LIN {X 0,Y 525.492,Z 369.575,A -85,B 0,C 180,E1 -4793.237,E2 -4793.237} C_VEL
LIN {X 0,Y 523.983,Z 361.217,A -85,B 0,C 180,E1 -4794.674,E2 -4794.674} C_VEL
LIN {X 0,Y 523.979,Z 361.219,A -85,B 0,C 180,E1 -4797.718,E2 -4797.718} C_VEL
LIN {X 0,Y 523.947,Z 361.217,A -85,B 0,C 180,E1 -4800.855,E2 -4800.855} C_VEL
LIN {X 0,Y 523.96,Z 361.222,A -85,B 0,C 180,E1 -4803.734,E2 -4803.734} C_VEL
LIN {X 0,Y 523.921,Z 361.218,A -85,B 0,C 180,E1 -4806.404,E2 -4806.404} C_VEL
LIN {X 0,Y 523.921,Z 361.22,A -85,B 0,C 180,E1 -4809.084,E2 -4809.084} C_VEL
LIN {X 0,Y 523.954,Z 361.216,A -85,B 0,C 180,E1 -4812.118,E2 -4812.118} C_VEL
LIN {X 0,Y 523.952,Z 361.219,A -85,B 0,C 180,E1 -4815.308,E2 -4815.308} C_VEL
LIN {X 0,Y 523.968,Z 361.212,A -85,B 0,C 180,E1 -4818.687,E2 -4818.687} C_VEL
LIN {X 0,Y 523.92,Z 361.221,A -85,B 0,C 180,E1 -4821.079,E2 -4821.079} C_VEL
LIN {X 0,Y 523.922,Z 361.221,A -85,B 0,C 180,E1 -4823.827,E2 -4823.827} C_VEL
LIN {X 0,Y 523.937,Z 361.216,A -85,B 0,C 180,E1 -4826.635,E2 -4826.635} C_VEL
LIN {X 0,Y 523.957,Z 361.223,A -85,B 0,C 180,E1 -4829.356,E2 -4829.356} C_VEL
LIN {X 0,Y 523.973,Z 361.211,A -85,B 0,C 180,E1 -4832.28,E2 -4832.28} C_VEL
LIN {X 0,Y 523.948,Z 361.215,A -85,B 0,C 180,E1 -4834.581,E2 -4834.581} C_VEL
LIN {X 0,Y 523.937,Z 361.223,A -85,B 0,C 180,E1 -4837.108,E2 -4837.108} C_VEL
LIN {X 0,Y 523.971,Z 361.213,A -85,B 0,C 180,E1 -4839.865,E2 -4839.865} C_VEL
LIN {X 0,Y 523.963,Z 361.217,A -85,B 0,C 180,E1 -4842.837,E2 -4842.837} C_VEL
LIN {X 0,Y 523.967,Z 361.22,A -85,B 0,C 180,E1 -4845.235,E2 -4845.235} C_VEL
LIN {X 0,Y 524.004,Z 361.208,A -85,B 0,C 180,E1 -4848.394,E2 -4848.394} C_VEL
LIN {X 0,Y 524,Z 361.211,A -85,B 0,C 180,E1 -4851.516,E2 -4851.516} C_VEL
LIN {X 0,Y 524.078,Z 361.202,A -85,B 0,C 180,E1 -4854.614,E2 -4854.614} C_VEL
LIN {X 0,Y 524.104,Z 361.196,A -85,B 0,C 180,E1 -4857.694,E2 -4857.694} C_VEL
LIN {X 0,Y 524.119,Z 361.2,A -85,B 0,C 180,E1 -4860.768,E2 -4860.768} C_VEL
LIN {X 0,Y 524.07,Z 361.206,A -85,B 0,C 180,E1 -4863.075,E2 -4863.075} C_VEL
LIN {X 0,Y 524.038,Z 361.204,A -85,B 0,C 180,E1 -4866.159,E2 -4866.159} C_VEL
LIN {X 0,Y 523.996,Z 361.211,A -85,B 0,C 180,E1 -4869.262,E2 -4869.262} C_VEL
LIN {X 0,Y 524.015,Z 361.206,A -85,B 0,C 180,E1 -4871.752,E2 -4871.752} C_VEL
LIN {X 0,Y 523.984,Z 361.214,A -85,B 0,C 180,E1 -4875.053,E2 -4875.053} C_VEL
LIN {X 0,Y 523.956,Z 361.214,A -85,B 0,C 180,E1 -4877.969,E2 -4877.969} C_VEL
LIN {X 0,Y 523.965,Z 361.218,A -85,B 0,C 180,E1 -4880.41,E2 -4880.41} C_VEL
LIN {X 0,Y 523.937,Z 361.221,A -85,B 0,C 180,E1 -4882.893,E2 -4882.893} C_VEL
LIN {X 0,Y 523.978,Z 361.212,A -85,B 0,C 180,E1 -4886.021,E2 -4886.021} C_VEL
LIN {X 0,Y 523.934,Z 361.221,A -85,B 0,C 180,E1 -4888.875,E2 -4888.875} C_VEL
LIN {X 0,Y 523.925,Z 361.217,A -85,B 0,C 180,E1 -4891.544,E2 -4891.544} C_VEL
LIN {X 0,Y 523.934,Z 361.223,A -85,B 0,C 180,E1 -4894.29,E2 -4894.29} C_VEL
LIN {X 0,Y 523.906,Z 361.22,A -85,B 0,C 180,E1 -4897.133,E2 -4897.133} C_VEL
LIN {X 0,Y 523.963,Z 361.218,A -85,B 0,C 180,E1 -4900.135,E2 -4900.135} C_VEL
LIN {X 0,Y 523.922,Z 361.218,A -85,B 0,C 180,E1 -4903.167,E2 -4903.167} C_VEL
LIN {X 0,Y 523.935,Z 361.218,A -85,B 0,C 180,E1 -4905.773,E2 -4905.773} C_VEL
LIN {X 0,Y 523.913,Z 361.22,A -85,B 0,C 180,E1 -4906.931,E2 -4906.931} C_VEL
LIN {X 0,Y 523.248,Z 361.303,A -85,B 0,C 180,E1 -4907.572,E2 -4907.572} C_VEL
LIN {X 0,Y 520.406,Z 361.666,A -85,B 0,C 180,E1 -4908.614,E2 -4908.614} C_VEL
LIN {X 0,Y 518,Z 361.971,A -85,B 0,C 180,E1 -4909.453,E2 -4909.453} C_VEL
LIN {X 0,Y 516.965,Z 362.096,A -85,B 0,C 180,E1 -4910.101,E2 -4910.101} C_VEL
LIN {X 0,Y 516.879,Z 362.103,A -85,B 0,C 180,E1 -4910.32,E2 -4910.32} C_VEL
LIN {X 0,Y 516.884,Z 362.095,A -85,B 0,C 180,E1 -4913.343,E2 -4913.343} C_VEL
LIN {X 0,Y 516.911,Z 362.1,A -85,B 0,C 180,E1 -4916.122,E2 -4916.122} C_VEL
LIN {X 0,Y 516.892,Z 362.094,A -85,B 0,C 180,E1 -4918.936,E2 -4918.936} C_VEL
LIN {X 0,Y 516.92,Z 362.092,A -85,B 0,C 180,E1 -4921.586,E2 -4921.586} C_VEL
LIN {X 0,Y 516.93,Z 362.097,A -85,B 0,C 180,E1 -4924.212,E2 -4924.212} C_VEL
LIN {X 0,Y 516.861,Z 362.101,A -85,B 0,C 180,E1 -4926.777,E2 -4926.777} C_VEL
LIN {X 0,Y 516.963,Z 362.173,A -85,B 0,C 180,E1 -4929.932,E2 -4929.932} C_VEL
LIN {X 0,Y 517.701,Z 368.131,A -85,B 0,C 180,E1 -4931.191,E2 -4931.191} C_VEL
LIN {X 0,Y 517.28,Z 383.258,A -85,B 0,C 180,E1 -4934.233,E2 -4934.233} C_VEL
LIN {X 0,Y 517.249,Z 385.513,A -85,B 0,C 180,E1 -4934.682,E2 -4934.682} C_VEL
LIN {X 0,Y 519.15,Z 395.792,A -85,B 0,C 180,E1 -4934.899,E2 -4934.899} C_VEL
LIN {X 0,Y 518.657,Z 492.288,A -85,B 0,C 180,E1 -4936.258,E2 -4936.258} C_VEL
LIN {X 0,Y 518.471,Z 505.449,A -85,B 0,C 180,E1 -4936.603,E2 -4936.603} C_VEL
LIN {X 0,Y 518.233,Z 517.533,A -85,B 0,C 180,E1 -4937.07,E2 -4937.07} C_VEL
LIN {X 0,Y 518.027,Z 528.523,A -85,B 0,C 180,E1 -4937.639,E2 -4937.639} C_VEL
LIN {X 0,Y 517.731,Z 539.307,A -85,B 0,C 180,E1 -4938.351,E2 -4938.351} C_VEL
LIN {X 0,Y 517.367,Z 549.993,A -85,B 0,C 180,E1 -4939.235,E2 -4939.235} C_VEL
LIN {X 0,Y 517.115,Z 559.603,A -85,B 0,C 180,E1 -4940.219,E2 -4940.219} C_VEL
LIN {X 0,Y 516.861,Z 567.474,A -85,B 0,C 180,E1 -4941.201,E2 -4941.201} C_VEL
LIN {X 0,Y 516.638,Z 575.169,A -85,B 0,C 180,E1 -4942.378,E2 -4942.378} C_VEL
LIN {X 0,Y 516.496,Z 582.223,A -85,B 0,C 180,E1 -4943.751,E2 -4943.751} C_VEL
LIN {X 0,Y 516.314,Z 586.928,A -85,B 0,C 180,E1 -4944.924,E2 -4944.924} C_VEL
LIN {X 0,Y 516.373,Z 590.524,A -85,B 0,C 180,E1 -4946.098,E2 -4946.098} C_VEL
LIN {X 0,Y 516.282,Z 592.387,A -85,B 0,C 180,E1 -4946.879,E2 -4946.879} C_VEL
LIN {X 0,Y 516.261,Z 593.792,A -85,B 0,C 180,E1 -4947.659,E2 -4947.659} C_VEL
LIN {X 0,Y 516.16,Z 595.409,A -85,B 0,C 180,E1 -4949.22,E2 -4949.22} C_VEL
LIN {X 0,Y 516.157,Z 595.646,A -85,B 0,C 180,E1 -4950,E2 -4950} C_VEL
LIN {X 0,Y 516.16,Z 595.463,A -85,B 0,C 180,E1 -4950.78,E2 -4950.78} C_VEL
LIN {X 0,Y 516.262,Z 593.917,A -85,B 0,C 180,E1 -4952.341,E2 -4952.341} C_VEL
LIN {X 0,Y 516.283,Z 592.567,A -85,B 0,C 180,E1 -4953.121,E2 -4953.121} C_VEL
LIN {X 0,Y 516.365,Z 589.71,A -85,B 0,C 180,E1 -4954.293,E2 -4954.293} C_VEL
LIN {X 0,Y 516.404,Z 585.839,A -85,B 0,C 180,E1 -4955.467,E2 -4955.467} C_VEL
LIN {X 0,Y 516.512,Z 580.842,A -85,B 0,C 180,E1 -4956.641,E2 -4956.641} C_VEL
LIN {X 0,Y 516.655,Z 574.551,A -85,B 0,C 180,E1 -4957.818,E2 -4957.818} C_VEL
LIN {X 0,Y 516.866,Z 566.672,A -85,B 0,C 180,E1 -4958.996,E2 -4958.996} C_VEL
LIN {X 0,Y 517.099,Z 558.64,A -85,B 0,C 180,E1 -4959.979,E2 -4959.979} C_VEL
LIN {X 0,Y 517.409,Z 548.833,A -85,B 0,C 180,E1 -4960.962,E2 -4960.962} C_VEL
LIN {X 0,Y 517.773,Z 538.044,A -85,B 0,C 180,E1 -4961.83,E2 -4961.83} C_VEL
LIN {X 0,Y 518.038,Z 527.003,A -85,B 0,C 180,E1 -4962.536,E2 -4962.536} C_VEL
LIN {X 0,Y 518.291,Z 515.07,A -85,B 0,C 180,E1 -4963.128,E2 -4963.128} C_VEL
LIN {X 0,Y 518.533,Z 502.017,A -85,B 0,C 180,E1 -4963.595,E2 -4963.595} C_VEL
LIN {X 0,Y 518.707,Z 488.929,A -85,B 0,C 180,E1 -4963.89,E2 -4963.89} C_VEL
LIN {X 0,Y 519.136,Z 396.282,A -85,B 0,C 180,E1 -4965.184,E2 -4965.184} C_VEL
LIN {X 0,Y 517.224,Z 385.584,A -85,B 0,C 180,E1 -4965.398,E2 -4965.398} C_VEL
LIN {X 0,Y 517.626,Z 370.592,A -85,B 0,C 180,E1 -4968.401,E2 -4968.401} C_VEL
LIN {X 0,Y 517.556,Z 365.569,A -85,B 0,C 180,E1 -4969.432,E2 -4969.432} C_VEL
LIN {X 0,Y 516.946,Z 362.096,A -85,B 0,C 180,E1 -4970.199,E2 -4970.199} C_VEL
LIN {X 0,Y 516.874,Z 362.102,A -85,B 0,C 180,E1 -4973.223,E2 -4973.223} C_VEL
LIN {X 0,Y 516.944,Z 362.093,A -85,B 0,C 180,E1 -4976.195,E2 -4976.195} C_VEL
LIN {X 0,Y 516.922,Z 362.091,A -85,B 0,C 180,E1 -4979.304,E2 -4979.304} C_VEL
LIN {X 0,Y 516.897,Z 362.094,A -85,B 0,C 180,E1 -4982.543,E2 -4982.543} C_VEL
LIN {X 0,Y 516.882,Z 362.097,A -85,B 0,C 180,E1 -4985.332,E2 -4985.332} C_VEL
LIN {X 0,Y 516.88,Z 362.103,A -85,B 0,C 180,E1 -4987.943,E2 -4987.943} C_VEL
LIN {X 0,Y 516.881,Z 362.095,A -85,B 0,C 180,E1 -4990.741,E2 -4990.741} C_VEL
LIN {X 0,Y 516.879,Z 362.095,A -85,B 0,C 180,E1 -4992.831,E2 -4992.831} C_VEL
LIN {X 0,Y 516.919,Z 362.091,A -85,B 0,C 180,E1 -4995.009,E2 -4995.009} C_VEL
LIN {X 0,Y 516.918,Z 362.091,A -85,B 0,C 180,E1 -4998.397,E2 -4998.397} C_VEL
LIN {X 0,Y 516.881,Z 362.099,A -85,B 0,C 180,E1 -5001.284,E2 -5001.284} C_VEL
LIN {X 0,Y 516.886,Z 362.096,A -85,B 0,C 180,E1 -5004.221,E2 -5004.221} C_VEL
LIN {X 0,Y 516.892,Z 362.096,A -85,B 0,C 180,E1 -5007.053,E2 -5007.053} C_VEL
LIN {X 0,Y 516.885,Z 362.099,A -85,B 0,C 180,E1 -5009.796,E2 -5009.796} C_VEL
LIN {X 0,Y 516.923,Z 362.09,A -85,B 0,C 180,E1 -5012.467,E2 -5012.467} C_VEL
LIN {X 0,Y 516.907,Z 362.095,A -85,B 0,C 180,E1 -5015.072,E2 -5015.072} C_VEL
LIN {X 0,Y 516.905,Z 362.098,A -85,B 0,C 180,E1 -5017.623,E2 -5017.623} C_VEL
LIN {X 0,Y 516.924,Z 362.09,A -85,B 0,C 180,E1 -5020.129,E2 -5020.129} C_VEL
LIN {X 0,Y 516.923,Z 362.09,A -85,B 0,C 180,E1 -5022.596,E2 -5022.596} C_VEL
LIN {X 0,Y 516.941,Z 362.092,A -85,B 0,C 180,E1 -5025.03,E2 -5025.03} C_VEL
LIN {X 0,Y 516.995,Z 362.081,A -85,B 0,C 180,E1 -5028.234,E2 -5028.234} C_VEL
LIN {X 0,Y 516.964,Z 362.091,A -85,B 0,C 180,E1 -5031.4,E2 -5031.4} C_VEL
LIN {X 0,Y 517.002,Z 362.082,A -85,B 0,C 180,E1 -5033.757,E2 -5033.757} C_VEL
LIN {X 0,Y 517.01,Z 362.084,A -85,B 0,C 180,E1 -5036.883,E2 -5036.883} C_VEL
LIN {X 0,Y 517.075,Z 362.071,A -85,B 0,C 180,E1 -5040,E2 -5040} C_VEL
LIN {X 0,Y 517.011,Z 362.087,A -85,B 0,C 180,E1 -5043.117,E2 -5043.117} C_VEL
LIN {X 0,Y 517.002,Z 362.08,A -85,B 0,C 180,E1 -5046.243,E2 -5046.243} C_VEL
LIN {X 0,Y 516.952,Z 362.089,A -85,B 0,C 180,E1 -5049.389,E2 -5049.389} C_VEL
LIN {X 0,Y 516.974,Z 362.083,A -85,B 0,C 180,E1 -5051.824,E2 -5051.824} C_VEL
LIN {X 0,Y 516.934,Z 362.093,A -85,B 0,C 180,E1 -5055.147,E2 -5055.147} C_VEL
LIN {X 0,Y 516.917,Z 362.092,A -85,B 0,C 180,E1 -5058.223,E2 -5058.223} C_VEL
LIN {X 0,Y 516.907,Z 362.099,A -85,B 0,C 180,E1 -5060.702,E2 -5060.702} C_VEL
LIN {X 0,Y 516.884,Z 362.097,A -85,B 0,C 180,E1 -5063.223,E2 -5063.223} C_VEL
LIN {X 0,Y 516.937,Z 362.09,A -85,B 0,C 180,E1 -5066.197,E2 -5066.197} C_VEL
LIN {X 0,Y 516.915,Z 362.092,A -85,B 0,C 180,E1 -5069.305,E2 -5069.305} C_VEL
LIN {X 0,Y 516.895,Z 362.101,A -85,B 0,C 180,E1 -5072.545,E2 -5072.545} C_VEL
LIN {X 0,Y 516.877,Z 362.096,A -85,B 0,C 180,E1 -5075.333,E2 -5075.333} C_VEL
LIN {X 0,Y 516.876,Z 362.097,A -85,B 0,C 180,E1 -5077.944,E2 -5077.944} C_VEL
LIN {X 0,Y 516.899,Z 362.098,A -85,B 0,C 180,E1 -5080.74,E2 -5080.74} C_VEL
LIN {X 0,Y 516.879,Z 362.097,A -85,B 0,C 180,E1 -5083.904,E2 -5083.904} C_VEL
LIN {X 0,Y 516.879,Z 362.099,A -85,B 0,C 180,E1 -5086.108,E2 -5086.108} C_VEL
LIN {X 0,Y 516.914,Z 362.1,A -85,B 0,C 180,E1 -5088.399,E2 -5088.399} C_VEL
LIN {X 0,Y 516.88,Z 362.095,A -85,B 0,C 180,E1 -5091.285,E2 -5091.285} C_VEL
LIN {X 0,Y 516.89,Z 362.101,A -85,B 0,C 180,E1 -5094.222,E2 -5094.222} C_VEL
LIN {X 0,Y 516.897,Z 362.093,A -85,B 0,C 180,E1 -5097.054,E2 -5097.054} C_VEL
LIN {X 0,Y 516.892,Z 362.096,A -85,B 0,C 180,E1 -5099.797,E2 -5099.797} C_VEL
LIN {X 0,Y 516.928,Z 362.096,A -85,B 0,C 180,E1 -5102.468,E2 -5102.468} C_VEL
LIN {X 0,Y 516.95,Z 362.193,A -85,B 0,C 180,E1 -5105.199,E2 -5105.199} C_VEL
LIN {X 0,Y 518.512,Z 370.662,A -85,B 0,C 180,E1 -5106.644,E2 -5106.644} C_VEL
LIN {X 0,Y 518.115,Z 386.391,A -85,B 0,C 180,E1 -5109.142,E2 -5109.142} C_VEL
LIN {X 0,Y 517.656,Z 406.191,A -85,B 0,C 180,E1 -5112.245,E2 -5112.245} C_VEL
LIN {X 0,Y 517.312,Z 421.636,A -85,B 0,C 180,E1 -5114.629,E2 -5114.629} C_VEL
LIN {X 0,Y 519.087,Z 434.195,A -85,B 0,C 180,E1 -5114.862,E2 -5114.862} C_VEL
LIN {X 0,Y 518.613,Z 529.97,A -85,B 0,C 180,E1 -5116.207,E2 -5116.207} C_VEL
LIN {X 0,Y 518.393,Z 543.256,A -85,B 0,C 180,E1 -5116.551,E2 -5116.551} C_VEL
LIN {X 0,Y 518.076,Z 556.556,A -85,B 0,C 180,E1 -5117.066,E2 -5117.066} C_VEL
LIN {X 0,Y 517.751,Z 568.906,A -85,B 0,C 180,E1 -5117.73,E2 -5117.73} C_VEL
LIN {X 0,Y 517.506,Z 580.636,A -85,B 0,C 180,E1 -5118.544,E2 -5118.544} C_VEL
LIN {X 0,Y 517.177,Z 590.844,A -85,B 0,C 180,E1 -5119.429,E2 -5119.429} C_VEL
LIN {X 0,Y 516.902,Z 600.033,A -85,B 0,C 180,E1 -5120.413,E2 -5120.413} C_VEL
LIN {X 0,Y 516.668,Z 608.989,A -85,B 0,C 180,E1 -5121.592,E2 -5121.592} C_VEL
LIN {X 0,Y 516.51,Z 616.199,A -85,B 0,C 180,E1 -5122.77,E2 -5122.77} C_VEL
LIN {X 0,Y 516.423,Z 622.768,A -85,B 0,C 180,E1 -5124.142,E2 -5124.142} C_VEL
LIN {X 0,Y 516.271,Z 627.109,A -85,B 0,C 180,E1 -5125.315,E2 -5125.315} C_VEL
LIN {X 0,Y 516.352,Z 629.413,A -85,B 0,C 180,E1 -5126.098,E2 -5126.098} C_VEL
LIN {X 0,Y 516.282,Z 631.276,A -85,B 0,C 180,E1 -5126.879,E2 -5126.879} C_VEL
LIN {X 0,Y 516.261,Z 632.674,A -85,B 0,C 180,E1 -5127.659,E2 -5127.659} C_VEL
LIN {X 0,Y 516.16,Z 634.277,A -85,B 0,C 180,E1 -5129.22,E2 -5129.22} C_VEL
LIN {X 0,Y 516.155,Z 634.494,A -85,B 0,C 180,E1 -5130,E2 -5130} C_VEL
LIN {X 0,Y 516.192,Z 633.671,A -85,B 0,C 180,E1 -5131.56,E2 -5131.56} C_VEL
LIN {X 0,Y 516.261,Z 632.677,A -85,B 0,C 180,E1 -5132.341,E2 -5132.341} C_VEL
LIN {X 0,Y 516.282,Z 631.28,A -85,B 0,C 180,E1 -5133.121,E2 -5133.121} C_VEL
LIN {X 0,Y 516.312,Z 628.34,A -85,B 0,C 180,E1 -5134.293,E2 -5134.293} C_VEL
LIN {X 0,Y 516.376,Z 624.361,A -85,B 0,C 180,E1 -5135.467,E2 -5135.467} C_VEL
LIN {X 0,Y 516.475,Z 618.48,A -85,B 0,C 180,E1 -5136.792,E2 -5136.792} C_VEL
LIN {X 0,Y 516.607,Z 611.554,A -85,B 0,C 180,E1 -5138.015,E2 -5138.015} C_VEL
LIN {X 0,Y 516.827,Z 603.259,A -85,B 0,C 180,E1 -5139.194,E2 -5139.194} C_VEL
LIN {X 0,Y 517.06,Z 594.759,A -85,B 0,C 180,E1 -5140.177,E2 -5140.177} C_VEL
LIN {X 0,Y 517.376,Z 584.258,A -85,B 0,C 180,E1 -5141.161,E2 -5141.161} C_VEL
LIN {X 0,Y 517.675,Z 573.086,A -85,B 0,C 180,E1 -5142.003,E2 -5142.003} C_VEL
LIN {X 0,Y 518.01,Z 562.49,A -85,B 0,C 180,E1 -5142.637,E2 -5142.637} C_VEL
LIN {X 0,Y 518.248,Z 550.819,A -85,B 0,C 180,E1 -5143.179,E2 -5143.179} C_VEL
LIN {X 0,Y 518.466,Z 537.374,A -85,B 0,C 180,E1 -5143.622,E2 -5143.622} C_VEL
LIN {X 0,Y 518.715,Z 524.11,A -85,B 0,C 180,E1 -5143.89,E2 -5143.89} C_VEL
LIN {X 0,Y 518.988,Z 432.488,A -85,B 0,C 180,E1 -5145.165,E2 -5145.165} C_VEL
LIN {X 0,Y 517.318,Z 421.613,A -85,B 0,C 180,E1 -5145.375,E2 -5145.375} C_VEL
LIN {X 0,Y 517.762,Z 400.778,A -85,B 0,C 180,E1 -5148.601,E2 -5148.601} C_VEL
LIN {X 0,Y 518.306,Z 382.467,A -85,B 0,C 180,E1 -5151.475,E2 -5151.475} C_VEL
LIN {X 0,Y 518.513,Z 370.659,A -85,B 0,C 180,E1 -5153.356,E2 -5153.356} C_VEL
LIN {X 0,Y 516.941,Z 362.094,A -85,B 0,C 180,E1 -5154.855,E2 -5154.855} C_VEL
LIN {X 0,Y 516.926,Z 362.097,A -85,B 0,C 180,E1 -5157.905,E2 -5157.905} C_VEL
LIN {X 0,Y 516.892,Z 362.099,A -85,B 0,C 180,E1 -5160.203,E2 -5160.203} C_VEL
LIN {X 0,Y 516.897,Z 362.093,A -85,B 0,C 180,E1 -5162.946,E2 -5162.946} C_VEL
LIN {X 0,Y 516.89,Z 362.101,A -85,B 0,C 180,E1 -5165.778,E2 -5165.778} C_VEL
LIN {X 0,Y 516.88,Z 362.095,A -85,B 0,C 180,E1 -5168.715,E2 -5168.715} C_VEL
LIN {X 0,Y 516.912,Z 362.097,A -85,B 0,C 180,E1 -5171.774,E2 -5171.774} C_VEL
LIN {X 0,Y 516.918,Z 362.092,A -85,B 0,C 180,E1 -5175.009,E2 -5175.009} C_VEL
LIN {X 0,Y 516.918,Z 362.09,A -85,B 0,C 180,E1 -5178.397,E2 -5178.397} C_VEL
LIN {X 0,Y 516.881,Z 362.101,A -85,B 0,C 180,E1 -5181.284,E2 -5181.284} C_VEL
LIN {X 0,Y 516.885,Z 362.095,A -85,B 0,C 180,E1 -5184.221,E2 -5184.221} C_VEL
LIN {X 0,Y 516.892,Z 362.098,A -85,B 0,C 180,E1 -5187.053,E2 -5187.053} C_VEL
LIN {X 0,Y 516.895,Z 362.096,A -85,B 0,C 180,E1 -5189.796,E2 -5189.796} C_VEL
LIN {X 0,Y 516.923,Z 362.09,A -85,B 0,C 180,E1 -5192.467,E2 -5192.467} C_VEL
LIN {X 0,Y 516.906,Z 362.098,A -85,B 0,C 180,E1 -5195.072,E2 -5195.072} C_VEL
LIN {X 0,Y 516.904,Z 362.096,A -85,B 0,C 180,E1 -5197.623,E2 -5197.623} C_VEL
LIN {X 0,Y 516.924,Z 362.089,A -85,B 0,C 180,E1 -5200.129,E2 -5200.129} C_VEL
LIN {X 0,Y 516.923,Z 362.091,A -85,B 0,C 180,E1 -5202.596,E2 -5202.596} C_VEL
LIN {X 0,Y 516.932,Z 362.096,A -85,B 0,C 180,E1 -5205.03,E2 -5205.03} C_VEL
LIN {X 0,Y 516.995,Z 362.081,A -85,B 0,C 180,E1 -5208.234,E2 -5208.234} C_VEL
LIN {X 0,Y 516.964,Z 362.089,A -85,B 0,C 180,E1 -5211.4,E2 -5211.4} C_VEL
LIN {X 0,Y 517.002,Z 362.08,A -85,B 0,C 180,E1 -5213.757,E2 -5213.757} C_VEL
LIN {X 0,Y 517.011,Z 362.086,A -85,B 0,C 180,E1 -5216.883,E2 -5216.883} C_VEL
LIN {X 0,Y 517.075,Z 362.071,A -85,B 0,C 180,E1 -5220,E2 -5220} C_VEL
LIN {X 0,Y 517.01,Z 362.085,A -85,B 0,C 180,E1 -5223.117,E2 -5223.117} C_VEL
LIN {X 0,Y 517.002,Z 362.081,A -85,B 0,C 180,E1 -5226.243,E2 -5226.243} C_VEL
LIN {X 0,Y 516.95,Z 362.088,A -85,B 0,C 180,E1 -5229.389,E2 -5229.389} C_VEL
LIN {X 0,Y 516.974,Z 362.083,A -85,B 0,C 180,E1 -5231.824,E2 -5231.824} C_VEL
LIN {X 0,Y 516.937,Z 362.091,A -85,B 0,C 180,E1 -5235.148,E2 -5235.148} C_VEL
LIN {X 0,Y 516.918,Z 362.093,A -85,B 0,C 180,E1 -5238.223,E2 -5238.223} C_VEL
LIN {X 0,Y 516.907,Z 362.1,A -85,B 0,C 180,E1 -5240.702,E2 -5240.702} C_VEL
LIN {X 0,Y 516.884,Z 362.096,A -85,B 0,C 180,E1 -5243.223,E2 -5243.223} C_VEL
LIN {X 0,Y 516.937,Z 362.091,A -85,B 0,C 180,E1 -5246.197,E2 -5246.197} C_VEL
LIN {X 0,Y 516.915,Z 362.091,A -85,B 0,C 180,E1 -5249.305,E2 -5249.305} C_VEL
LIN {X 0,Y 516.894,Z 362.102,A -85,B 0,C 180,E1 -5252.545,E2 -5252.545} C_VEL
LIN {X 0,Y 516.873,Z 362.096,A -85,B 0,C 180,E1 -5255.333,E2 -5255.333} C_VEL
LIN {X 0,Y 516.877,Z 362.098,A -85,B 0,C 180,E1 -5257.944,E2 -5257.944} C_VEL
LIN {X 0,Y 516.899,Z 362.096,A -85,B 0,C 180,E1 -5260.74,E2 -5260.74} C_VEL
LIN {X 0,Y 516.879,Z 362.098,A -85,B 0,C 180,E1 -5263.904,E2 -5263.904} C_VEL
LIN {X 0,Y 516.878,Z 362.101,A -85,B 0,C 180,E1 -5266.108,E2 -5266.108} C_VEL
LIN {X 0,Y 516.912,Z 362.098,A -85,B 0,C 180,E1 -5268.399,E2 -5268.399} C_VEL
LIN {X 0,Y 516.879,Z 362.103,A -85,B 0,C 180,E1 -5270.32,E2 -5270.32} C_VEL
LIN {X 0,Y 516.21,Z 362.181,A -85,B 0,C 180,E1 -5270.97,E2 -5270.97} C_VEL
LIN {X 0,Y 513.364,Z 362.539,A -85,B 0,C 180,E1 -5272.026,E2 -5272.026} C_VEL
LIN {X 0,Y 510.956,Z 362.837,A -85,B 0,C 180,E1 -5272.877,E2 -5272.877} C_VEL
LIN {X 0,Y 509.917,Z 362.964,A -85,B 0,C 180,E1 -5273.533,E2 -5273.533} C_VEL
LIN {X 0,Y 509.83,Z 362.975,A -85,B 0,C 180,E1 -5273.756,E2 -5273.756} C_VEL
LIN {X 0,Y 509.861,Z 362.973,A -85,B 0,C 180,E1 -5276.54,E2 -5276.54} C_VEL
LIN {X 0,Y 509.849,Z 362.971,A -85,B 0,C 180,E1 -5279.335,E2 -5279.335} C_VEL
LIN {X 0,Y 509.894,Z 362.974,A -85,B 0,C 180,E1 -5282.055,E2 -5282.055} C_VEL
LIN {X 0,Y 509.841,Z 362.976,A -85,B 0,C 180,E1 -5284.703,E2 -5284.703} C_VEL
LIN {X 0,Y 509.828,Z 362.978,A -85,B 0,C 180,E1 -5287.459,E2 -5287.459} C_VEL
LIN {X 0,Y 509.921,Z 362.997,A -85,B 0,C 180,E1 -5289.771,E2 -5289.771} C_VEL
LIN {X 0,Y 510.746,Z 369.35,A -85,B 0,C 180,E1 -5291.134,E2 -5291.134} C_VEL
LIN {X 0,Y 510.264,Z 384.704,A -85,B 0,C 180,E1 -5294.257,E2 -5294.257} C_VEL
LIN {X 0,Y 510.243,Z 385.813,A -85,B 0,C 180,E1 -5294.479,E2 -5294.479} C_VEL
LIN {X 0,Y 512.337,Z 397.539,A -85,B 0,C 180,E1 -5294.714,E2 -5294.714} C_VEL
LIN {X 0,Y 511.79,Z 492.582,A -85,B 0,C 180,E1 -5296.07,E2 -5296.07} C_VEL
LIN {X 0,Y 511.572,Z 505.735,A -85,B 0,C 180,E1 -5296.418,E2 -5296.418} C_VEL
LIN {X 0,Y 511.342,Z 517.814,A -85,B 0,C 180,E1 -5296.893,E2 -5296.893} C_VEL
LIN {X 0,Y 511.105,Z 529.323,A -85,B 0,C 180,E1 -5297.5,E2 -5297.5} C_VEL
LIN {X 0,Y 510.749,Z 540.867,A -85,B 0,C 180,E1 -5298.29,E2 -5298.29} C_VEL
LIN {X 0,Y 510.363,Z 551.331,A -85,B 0,C 180,E1 -5299.186,E2 -5299.186} C_VEL
LIN {X 0,Y 510.107,Z 559.876,A -85,B 0,C 180,E1 -5300.083,E2 -5300.083} C_VEL
LIN {X 0,Y 509.856,Z 567.745,A -85,B 0,C 180,E1 -5301.079,E2 -5301.079} C_VEL
LIN {X 0,Y 509.611,Z 575.439,A -85,B 0,C 180,E1 -5302.273,E2 -5302.273} C_VEL
LIN {X 0,Y 509.431,Z 582.493,A -85,B 0,C 180,E1 -5303.664,E2 -5303.664} C_VEL
LIN {X 0,Y 509.248,Z 587.197,A -85,B 0,C 180,E1 -5304.854,E2 -5304.854} C_VEL
LIN {X 0,Y 509.304,Z 590.792,A -85,B 0,C 180,E1 -5306.044,E2 -5306.044} C_VEL
LIN {X 0,Y 509.201,Z 592.656,A -85,B 0,C 180,E1 -5306.835,E2 -5306.835} C_VEL
LIN {X 0,Y 509.19,Z 594.059,A -85,B 0,C 180,E1 -5307.627,E2 -5307.627} C_VEL
LIN {X 0,Y 509.074,Z 595.676,A -85,B 0,C 180,E1 -5309.209,E2 -5309.209} C_VEL
LIN {X 0,Y 509.068,Z 595.912,A -85,B 0,C 180,E1 -5310,E2 -5310} C_VEL
LIN {X 0,Y 509.074,Z 595.729,A -85,B 0,C 180,E1 -5310.791,E2 -5310.791} C_VEL
LIN {X 0,Y 509.19,Z 594.183,A -85,B 0,C 180,E1 -5312.373,E2 -5312.373} C_VEL
LIN {X 0,Y 509.202,Z 592.833,A -85,B 0,C 180,E1 -5313.165,E2 -5313.165} C_VEL
LIN {X 0,Y 509.289,Z 589.976,A -85,B 0,C 180,E1 -5314.353,E2 -5314.353} C_VEL
LIN {X 0,Y 509.348,Z 586.103,A -85,B 0,C 180,E1 -5315.542,E2 -5315.542} C_VEL
LIN {X 0,Y 509.488,Z 580.348,A -85,B 0,C 180,E1 -5316.891,E2 -5316.891} C_VEL
LIN {X 0,Y 509.646,Z 573.594,A -85,B 0,C 180,E1 -5318.126,E2 -5318.126} C_VEL
LIN {X 0,Y 509.908,Z 565.458,A -85,B 0,C 180,E1 -5319.32,E2 -5319.32} C_VEL
LIN {X 0,Y 510.135,Z 557.131,A -85,B 0,C 180,E1 -5320.317,E2 -5320.317} C_VEL
LIN {X 0,Y 510.523,Z 546.843,A -85,B 0,C 180,E1 -5321.313,E2 -5321.313} C_VEL
LIN {X 0,Y 510.893,Z 535.347,A -85,B 0,C 180,E1 -5322.202,E2 -5322.202} C_VEL
LIN {X 0,Y 511.212,Z 523.687,A -85,B 0,C 180,E1 -5322.909,E2 -5322.909} C_VEL
LIN {X 0,Y 511.477,Z 511.676,A -85,B 0,C 180,E1 -5323.458,E2 -5323.458} C_VEL
LIN {X 0,Y 511.712,Z 498.604,A -85,B 0,C 180,E1 -5323.882,E2 -5323.882} C_VEL
LIN {X 0,Y 511.821,Z 486.095,A -85,B 0,C 180,E1 -5324.132,E2 -5324.132} C_VEL
LIN {X 0,Y 512.279,Z 396.67,A -85,B 0,C 180,E1 -5325.39,E2 -5325.39} C_VEL
LIN {X 0,Y 510.259,Z 385.743,A -85,B 0,C 180,E1 -5325.628,E2 -5325.628} C_VEL
LIN {X 0,Y 510.693,Z 370.798,A -85,B 0,C 180,E1 -5328.66,E2 -5328.66} C_VEL
LIN {X 0,Y 510.584,Z 366.781,A -85,B 0,C 180,E1 -5329.499,E2 -5329.499} C_VEL
LIN {X 0,Y 509.909,Z 362.973,A -85,B 0,C 180,E1 -5330.344,E2 -5330.344} C_VEL
LIN {X 0,Y 509.839,Z 362.981,A -85,B 0,C 180,E1 -5333.562,E2 -5333.562} C_VEL
LIN {X 0,Y 509.912,Z 362.967,A -85,B 0,C 180,E1 -5336.378,E2 -5336.378} C_VEL
LIN {X 0,Y 509.877,Z 362.967,A -85,B 0,C 180,E1 -5338.843,E2 -5338.843} C_VEL
LIN {X 0,Y 509.822,Z 362.978,A -85,B 0,C 180,E1 -5341.589,E2 -5341.589} C_VEL
LIN {X 0,Y 509.853,Z 362.973,A -85,B 0,C 180,E1 -5344.412,E2 -5344.412} C_VEL
LIN {X 0,Y 509.818,Z 362.977,A -85,B 0,C 180,E1 -5347.34,E2 -5347.34} C_VEL
LIN {X 0,Y 509.835,Z 362.974,A -85,B 0,C 180,E1 -5350.381,E2 -5350.381} C_VEL
LIN {X 0,Y 509.819,Z 362.975,A -85,B 0,C 180,E1 -5353.061,E2 -5353.061} C_VEL
LIN {X 0,Y 509.827,Z 362.982,A -85,B 0,C 180,E1 -5355.791,E2 -5355.791} C_VEL
LIN {X 0,Y 509.861,Z 362.969,A -85,B 0,C 180,E1 -5358.575,E2 -5358.575} C_VEL
LIN {X 0,Y 509.847,Z 362.978,A -85,B 0,C 180,E1 -5361.785,E2 -5361.785} C_VEL
LIN {X 0,Y 509.841,Z 362.972,A -85,B 0,C 180,E1 -5364.623,E2 -5364.623} C_VEL
LIN {X 0,Y 509.86,Z 362.977,A -85,B 0,C 180,E1 -5367.481,E2 -5367.481} C_VEL
LIN {X 0,Y 509.851,Z 362.971,A -85,B 0,C 180,E1 -5370.273,E2 -5370.273} C_VEL
LIN {X 0,Y 509.88,Z 362.969,A -85,B 0,C 180,E1 -5372.944,E2 -5372.944} C_VEL
LIN {X 0,Y 509.868,Z 362.976,A -85,B 0,C 180,E1 -5375.574,E2 -5375.574} C_VEL
LIN {X 0,Y 509.841,Z 362.972,A -85,B 0,C 180,E1 -5378.149,E2 -5378.149} C_VEL
LIN {X 0,Y 509.857,Z 362.971,A -85,B 0,C 180,E1 -5380.681,E2 -5380.681} C_VEL
LIN {X 0,Y 509.88,Z 362.973,A -85,B 0,C 180,E1 -5383.174,E2 -5383.174} C_VEL
LIN {X 0,Y 509.865,Z 362.973,A -85,B 0,C 180,E1 -5385.634,E2 -5385.634} C_VEL
LIN {X 0,Y 509.917,Z 362.966,A -85,B 0,C 180,E1 -5388.875,E2 -5388.875} C_VEL
LIN {X 0,Y 509.943,Z 362.959,A -85,B 0,C 180,E1 -5392.078,E2 -5392.078} C_VEL
LIN {X 0,Y 509.976,Z 362.956,A -85,B 0,C 180,E1 -5394.464,E2 -5394.464} C_VEL
LIN {X 0,Y 510.047,Z 362.949,A -85,B 0,C 180,E1 -5397.631,E2 -5397.631} C_VEL
LIN {X 0,Y 510.058,Z 362.949,A -85,B 0,C 180,E1 -5400.789,E2 -5400.789} C_VEL
LIN {X 0,Y 509.953,Z 362.965,A -85,B 0,C 180,E1 -5403.16,E2 -5403.16} C_VEL
LIN {X 0,Y 509.97,Z 362.957,A -85,B 0,C 180,E1 -5406.33,E2 -5406.33} C_VEL
LIN {X 0,Y 509.911,Z 362.968,A -85,B 0,C 180,E1 -5408.72,E2 -5408.72} C_VEL
LIN {X 0,Y 509.942,Z 362.959,A -85,B 0,C 180,E1 -5411.931,E2 -5411.931} C_VEL
LIN {X 0,Y 509.884,Z 362.97,A -85,B 0,C 180,E1 -5415.242,E2 -5415.242} C_VEL
LIN {X 0,Y 509.88,Z 362.967,A -85,B 0,C 180,E1 -5418.001,E2 -5418.001} C_VEL
LIN {X 0,Y 509.849,Z 362.977,A -85,B 0,C 180,E1 -5421.002,E2 -5421.002} C_VEL
LIN {X 0,Y 509.843,Z 362.972,A -85,B 0,C 180,E1 -5423.563,E2 -5423.563} C_VEL
LIN {X 0,Y 509.906,Z 362.968,A -85,B 0,C 180,E1 -5426.38,E2 -5426.38} C_VEL
LIN {X 0,Y 509.87,Z 362.975,A -85,B 0,C 180,E1 -5428.845,E2 -5428.845} C_VEL
LIN {X 0,Y 509.818,Z 362.975,A -85,B 0,C 180,E1 -5431.59,E2 -5431.59} C_VEL
LIN {X 0,Y 509.848,Z 362.977,A -85,B 0,C 180,E1 -5434.414,E2 -5434.414} C_VEL
LIN {X 0,Y 509.813,Z 362.976,A -85,B 0,C 180,E1 -5437.341,E2 -5437.341} C_VEL
LIN {X 0,Y 509.856,Z 362.977,A -85,B 0,C 180,E1 -5440.381,E2 -5440.381} C_VEL
LIN {X 0,Y 509.835,Z 362.974,A -85,B 0,C 180,E1 -5443.065,E2 -5443.065} C_VEL
LIN {X 0,Y 509.826,Z 362.975,A -85,B 0,C 180,E1 -5445.793,E2 -5445.793} C_VEL
LIN {X 0,Y 509.855,Z 362.977,A -85,B 0,C 180,E1 -5448.576,E2 -5448.576} C_VEL
LIN {X 0,Y 509.849,Z 362.972,A -85,B 0,C 180,E1 -5451.787,E2 -5451.787} C_VEL
LIN {X 0,Y 509.845,Z 362.976,A -85,B 0,C 180,E1 -5454.624,E2 -5454.624} C_VEL
LIN {X 0,Y 509.865,Z 362.969,A -85,B 0,C 180,E1 -5457.482,E2 -5457.482} C_VEL
LIN {X 0,Y 509.858,Z 362.979,A -85,B 0,C 180,E1 -5460.274,E2 -5460.274} C_VEL
LIN {X 0,Y 509.885,Z 362.972,A -85,B 0,C 180,E1 -5462.945,E2 -5462.945} C_VEL
LIN {X 0,Y 509.923,Z 363.082,A -85,B 0,C 180,E1 -5465.018,E2 -5465.018} C_VEL
LIN {X 0,Y 511.538,Z 371.743,A -85,B 0,C 180,E1 -5466.521,E2 -5466.521} C_VEL
LIN {X 0,Y 511.238,Z 386.16,A -85,B 0,C 180,E1 -5468.848,E2 -5468.848} C_VEL
LIN {X 0,Y 510.648,Z 407.336,A -85,B 0,C 180,E1 -5472.211,E2 -5472.211} C_VEL
LIN {X 0,Y 510.314,Z 421.386,A -85,B 0,C 180,E1 -5474.417,E2 -5474.417} C_VEL
LIN {X 0,Y 512.226,Z 435.057,A -85,B 0,C 180,E1 -5474.671,E2 -5474.671} C_VEL
LIN {X 0,Y 511.727,Z 529.703,A -85,B 0,C 180,E1 -5476.018,E2 -5476.018} C_VEL
LIN {X 0,Y 511.483,Z 542.989,A -85,B 0,C 180,E1 -5476.365,E2 -5476.365} C_VEL
LIN {X 0,Y 511.154,Z 556.289,A -85,B 0,C 180,E1 -5476.888,E2 -5476.888} C_VEL
LIN {X 0,Y 510.837,Z 567.961,A -85,B 0,C 180,E1 -5477.518,E2 -5477.518} C_VEL
LIN {X 0,Y 510.55,Z 579.07,A -85,B 0,C 180,E1 -5478.285,E2 -5478.285} C_VEL
LIN {X 0,Y 510.242,Z 589.531,A -85,B 0,C 180,E1 -5479.184,E2 -5479.184} C_VEL
LIN {X 0,Y 509.94,Z 598.083,A -85,B 0,C 180,E1 -5480.08,E2 -5480.08} C_VEL
LIN {X 0,Y 509.694,Z 605.977,A -85,B 0,C 180,E1 -5481.076,E2 -5481.076} C_VEL
LIN {X 0,Y 509.484,Z 613.688,A -85,B 0,C 180,E1 -5482.271,E2 -5482.271} C_VEL
LIN {X 0,Y 509.319,Z 619.928,A -85,B 0,C 180,E1 -5483.473,E2 -5483.473} C_VEL
LIN {X 0,Y 509.243,Z 625.529,A -85,B 0,C 180,E1 -5484.853,E2 -5484.853} C_VEL
LIN {X 0,Y 509.246,Z 629.145,A -85,B 0,C 180,E1 -5486.043,E2 -5486.043} C_VEL
LIN {X 0,Y 509.2,Z 631.009,A -85,B 0,C 180,E1 -5486.835,E2 -5486.835} C_VEL
LIN {X 0,Y 509.189,Z 632.408,A -85,B 0,C 180,E1 -5487.627,E2 -5487.627} C_VEL
LIN {X 0,Y 509.073,Z 634.011,A -85,B 0,C 180,E1 -5489.209,E2 -5489.209} C_VEL
LIN {X 0,Y 509.066,Z 634.227,A -85,B 0,C 180,E1 -5490,E2 -5490} C_VEL
LIN {X 0,Y 509.112,Z 633.405,A -85,B 0,C 180,E1 -5491.582,E2 -5491.582} C_VEL
LIN {X 0,Y 509.189,Z 632.411,A -85,B 0,C 180,E1 -5492.373,E2 -5492.373} C_VEL
LIN {X 0,Y 509.2,Z 631.013,A -85,B 0,C 180,E1 -5493.165,E2 -5493.165} C_VEL
LIN {X 0,Y 509.205,Z 628.072,A -85,B 0,C 180,E1 -5494.353,E2 -5494.353} C_VEL
LIN {X 0,Y 509.294,Z 624.093,A -85,B 0,C 180,E1 -5495.543,E2 -5495.543} C_VEL
LIN {X 0,Y 509.407,Z 618.075,A -85,B 0,C 180,E1 -5496.914,E2 -5496.914} C_VEL
LIN {X 0,Y 509.551,Z 611.286,A -85,B 0,C 180,E1 -5498.127,E2 -5498.127} C_VEL
LIN {X 0,Y 509.764,Z 602.99,A -85,B 0,C 180,E1 -5499.322,E2 -5499.322} C_VEL
LIN {X 0,Y 510.028,Z 594.49,A -85,B 0,C 180,E1 -5500.319,E2 -5500.319} C_VEL
LIN {X 0,Y 510.387,Z 583.99,A -85,B 0,C 180,E1 -5501.316,E2 -5501.316} C_VEL
LIN {X 0,Y 510.67,Z 573.676,A -85,B 0,C 180,E1 -5502.11,E2 -5502.11} C_VEL
LIN {X 0,Y 511.056,Z 562.222,A -85,B 0,C 180,E1 -5502.812,E2 -5502.812} C_VEL
LIN {X 0,Y 511.32,Z 550.551,A -85,B 0,C 180,E1 -5503.361,E2 -5503.361} C_VEL
LIN {X 0,Y 511.571,Z 537.107,A -85,B 0,C 180,E1 -5503.809,E2 -5503.809} C_VEL
LIN {X 0,Y 511.84,Z 523.843,A -85,B 0,C 180,E1 -5504.081,E2 -5504.081} C_VEL
LIN {X 0,Y 512.175,Z 433.563,A -85,B 0,C 180,E1 -5505.352,E2 -5505.352} C_VEL
LIN {X 0,Y 510.301,Z 421.303,A -85,B 0,C 180,E1 -5505.598,E2 -5505.598} C_VEL
LIN {X 0,Y 510.762,Z 401.853,A -85,B 0,C 180,E1 -5508.657,E2 -5508.657} C_VEL
LIN {X 0,Y 511.364,Z 383.544,A -85,B 0,C 180,E1 -5511.57,E2 -5511.57} C_VEL
LIN {X 0,Y 511.539,Z 371.739,A -85,B 0,C 180,E1 -5513.479,E2 -5513.479} C_VEL
LIN {X 0,Y 509.898,Z 362.972,A -85,B 0,C 180,E1 -5515.007,E2 -5515.007} C_VEL
LIN {X 0,Y 509.898,Z 362.972,A -85,B 0,C 180,E1 -5518.1,E2 -5518.1} C_VEL
LIN {X 0,Y 509.847,Z 362.977,A -85,B 0,C 180,E1 -5521.28,E2 -5521.28} C_VEL
LIN {X 0,Y 509.86,Z 362.972,A -85,B 0,C 180,E1 -5524.203,E2 -5524.203} C_VEL
LIN {X 0,Y 509.817,Z 362.979,A -85,B 0,C 180,E1 -5527.34,E2 -5527.34} C_VEL
LIN {X 0,Y 509.836,Z 362.973,A -85,B 0,C 180,E1 -5530.381,E2 -5530.381} C_VEL
LIN {X 0,Y 509.836,Z 362.975,A -85,B 0,C 180,E1 -5533.063,E2 -5533.063} C_VEL
LIN {X 0,Y 509.827,Z 362.979,A -85,B 0,C 180,E1 -5535.791,E2 -5535.791} C_VEL
LIN {X 0,Y 509.861,Z 362.969,A -85,B 0,C 180,E1 -5538.575,E2 -5538.575} C_VEL
LIN {X 0,Y 509.847,Z 362.975,A -85,B 0,C 180,E1 -5541.785,E2 -5541.785} C_VEL
LIN {X 0,Y 509.84,Z 362.972,A -85,B 0,C 180,E1 -5544.623,E2 -5544.623} C_VEL
LIN {X 0,Y 509.86,Z 362.977,A -85,B 0,C 180,E1 -5547.481,E2 -5547.481} C_VEL
LIN {X 0,Y 509.875,Z 362.968,A -85,B 0,C 180,E1 -5550.268,E2 -5550.268} C_VEL
LIN {X 0,Y 509.88,Z 362.971,A -85,B 0,C 180,E1 -5552.944,E2 -5552.944} C_VEL
LIN {X 0,Y 509.867,Z 362.973,A -85,B 0,C 180,E1 -5555.574,E2 -5555.574} C_VEL
LIN {X 0,Y 509.841,Z 362.972,A -85,B 0,C 180,E1 -5558.149,E2 -5558.149} C_VEL
LIN {X 0,Y 509.857,Z 362.972,A -85,B 0,C 180,E1 -5560.681,E2 -5560.681} C_VEL
LIN {X 0,Y 509.879,Z 362.976,A -85,B 0,C 180,E1 -5563.175,E2 -5563.175} C_VEL
LIN {X 0,Y 509.855,Z 362.972,A -85,B 0,C 180,E1 -5565.634,E2 -5565.634} C_VEL
LIN {X 0,Y 509.92,Z 362.968,A -85,B 0,C 180,E1 -5568.875,E2 -5568.875} C_VEL
LIN {X 0,Y 509.943,Z 362.959,A -85,B 0,C 180,E1 -5572.078,E2 -5572.078} C_VEL
LIN {X 0,Y 509.976,Z 362.957,A -85,B 0,C 180,E1 -5574.464,E2 -5574.464} C_VEL
LIN {X 0,Y 510.047,Z 362.947,A -85,B 0,C 180,E1 -5577.631,E2 -5577.631} C_VEL
LIN {X 0,Y 510.058,Z 362.952,A -85,B 0,C 180,E1 -5580.79,E2 -5580.79} C_VEL
LIN {X 0,Y 509.953,Z 362.963,A -85,B 0,C 180,E1 -5583.16,E2 -5583.16} C_VEL
LIN {X 0,Y 509.97,Z 362.958,A -85,B 0,C 180,E1 -5586.33,E2 -5586.33} C_VEL
LIN {X 0,Y 509.911,Z 362.971,A -85,B 0,C 180,E1 -5588.72,E2 -5588.72} C_VEL
LIN {X 0,Y 509.942,Z 362.959,A -85,B 0,C 180,E1 -5591.931,E2 -5591.931} C_VEL
LIN {X 0,Y 509.884,Z 362.969,A -85,B 0,C 180,E1 -5595.242,E2 -5595.242} C_VEL
LIN {X 0,Y 509.88,Z 362.968,A -85,B 0,C 180,E1 -5598.002,E2 -5598.002} C_VEL
LIN {X 0,Y 509.849,Z 362.975,A -85,B 0,C 180,E1 -5601.002,E2 -5601.002} C_VEL
LIN {X 0,Y 509.843,Z 362.972,A -85,B 0,C 180,E1 -5603.563,E2 -5603.563} C_VEL
LIN {X 0,Y 509.906,Z 362.97,A -85,B 0,C 180,E1 -5606.38,E2 -5606.38} C_VEL
LIN {X 0,Y 509.87,Z 362.973,A -85,B 0,C 180,E1 -5608.845,E2 -5608.845} C_VEL
LIN {X 0,Y 509.819,Z 362.975,A -85,B 0,C 180,E1 -5611.59,E2 -5611.59} C_VEL
LIN {X 0,Y 509.846,Z 362.98,A -85,B 0,C 180,E1 -5614.414,E2 -5614.414} C_VEL
LIN {X 0,Y 509.814,Z 362.975,A -85,B 0,C 180,E1 -5617.341,E2 -5617.341} C_VEL
LIN {X 0,Y 509.857,Z 362.979,A -85,B 0,C 180,E1 -5620.381,E2 -5620.381} C_VEL
LIN {X 0,Y 509.836,Z 362.973,A -85,B 0,C 180,E1 -5623.065,E2 -5623.065} C_VEL
LIN {X 0,Y 509.826,Z 362.976,A -85,B 0,C 180,E1 -5625.793,E2 -5625.793} C_VEL
LIN {X 0,Y 509.853,Z 362.975,A -85,B 0,C 180,E1 -5628.575,E2 -5628.575} C_VEL
LIN {X 0,Y 509.85,Z 362.974,A -85,B 0,C 180,E1 -5631.787,E2 -5631.787} C_VEL
LIN {X 0,Y 509.83,Z 362.975,A -85,B 0,C 180,E1 -5633.756,E2 -5633.756} C_VEL
LIN {X 0,Y 509.165,Z 363.062,A -85,B 0,C 180,E1 -5634.415,E2 -5634.415} C_VEL
LIN {X 0,Y 506.347,Z 363.408,A -85,B 0,C 180,E1 -5635.487,E2 -5635.487} C_VEL
LIN {X 0,Y 503.953,Z 363.712,A -85,B 0,C 180,E1 -5636.35,E2 -5636.35} C_VEL
LIN {X 0,Y 502.903,Z 363.837,A -85,B 0,C 180,E1 -5637.017,E2 -5637.017} C_VEL
LIN {X 0,Y 502.806,Z 363.848,A -85,B 0,C 180,E1 -5637.242,E2 -5637.242} C_VEL
LIN {X 0,Y 502.816,Z 363.855,A -85,B 0,C 180,E1 -5640.065,E2 -5640.065} C_VEL
LIN {X 0,Y 502.834,Z 363.848,A -85,B 0,C 180,E1 -5642.534,E2 -5642.534} C_VEL
LIN {X 0,Y 502.804,Z 363.852,A -85,B 0,C 180,E1 -5645.306,E2 -5645.306} C_VEL
LIN {X 0,Y 502.781,Z 363.86,A -85,B 0,C 180,E1 -5647.827,E2 -5647.827} C_VEL
LIN {X 0,Y 502.872,Z 363.943,A -85,B 0,C 180,E1 -5649.63,E2 -5649.63} C_VEL
LIN {X 0,Y 503.766,Z 370.571,A -85,B 0,C 180,E1 -5651.074,E2 -5651.074} C_VEL
LIN {X 0,Y 503.278,Z 385.956,A -85,B 0,C 180,E1 -5654.237,E2 -5654.237} C_VEL
LIN {X 0,Y 505.494,Z 398.244,A -85,B 0,C 180,E1 -5654.508,E2 -5654.508} C_VEL
LIN {X 0,Y 504.926,Z 492.878,A -85,B 0,C 180,E1 -5655.877,E2 -5655.877} C_VEL
LIN {X 0,Y 504.679,Z 506.022,A -85,B 0,C 180,E1 -5656.229,E2 -5656.229} C_VEL
LIN {X 0,Y 504.441,Z 518.095,A -85,B 0,C 180,E1 -5656.71,E2 -5656.71} C_VEL
LIN {X 0,Y 504.192,Z 528.365,A -85,B 0,C 180,E1 -5657.253,E2 -5657.253} C_VEL
LIN {X 0,Y 503.854,Z 539.857,A -85,B 0,C 180,E1 -5658.025,E2 -5658.025} C_VEL
LIN {X 0,Y 503.448,Z 550.54,A -85,B 0,C 180,E1 -5658.934,E2 -5658.934} C_VEL
LIN {X 0,Y 503.121,Z 560.148,A -85,B 0,C 180,E1 -5659.944,E2 -5659.944} C_VEL
LIN {X 0,Y 502.851,Z 568.017,A -85,B 0,C 180,E1 -5660.954,E2 -5660.954} C_VEL
LIN {X 0,Y 502.571,Z 575.71,A -85,B 0,C 180,E1 -5662.164,E2 -5662.164} C_VEL
LIN {X 0,Y 502.362,Z 582.763,A -85,B 0,C 180,E1 -5663.574,E2 -5663.574} C_VEL
LIN {X 0,Y 502.187,Z 587.466,A -85,B 0,C 180,E1 -5664.781,E2 -5664.781} C_VEL
LIN {X 0,Y 502.237,Z 591.06,A -85,B 0,C 180,E1 -5665.988,E2 -5665.988} C_VEL
LIN {X 0,Y 502.124,Z 592.924,A -85,B 0,C 180,E1 -5666.791,E2 -5666.791} C_VEL
LIN {X 0,Y 502.121,Z 594.326,A -85,B 0,C 180,E1 -5667.594,E2 -5667.594} C_VEL
LIN {X 0,Y 501.991,Z 595.943,A -85,B 0,C 180,E1 -5669.198,E2 -5669.198} C_VEL
LIN {X 0,Y 501.983,Z 596.179,A -85,B 0,C 180,E1 -5670,E2 -5670} C_VEL
LIN {X 0,Y 501.99,Z 595.995,A -85,B 0,C 180,E1 -5670.802,E2 -5670.802} C_VEL
LIN {X 0,Y 502.121,Z 594.448,A -85,B 0,C 180,E1 -5672.406,E2 -5672.406} C_VEL
LIN {X 0,Y 502.125,Z 593.098,A -85,B 0,C 180,E1 -5673.209,E2 -5673.209} C_VEL
LIN {X 0,Y 502.214,Z 590.241,A -85,B 0,C 180,E1 -5674.414,E2 -5674.414} C_VEL
LIN {X 0,Y 502.294,Z 586.368,A -85,B 0,C 180,E1 -5675.621,E2 -5675.621} C_VEL
LIN {X 0,Y 502.402,Z 581.371,A -85,B 0,C 180,E1 -5676.828,E2 -5676.828} C_VEL
LIN {X 0,Y 502.574,Z 575.079,A -85,B 0,C 180,E1 -5678.038,E2 -5678.038} C_VEL
LIN {X 0,Y 502.819,Z 567.198,A -85,B 0,C 180,E1 -5679.25,E2 -5679.25} C_VEL
LIN {X 0,Y 503.119,Z 559.163,A -85,B 0,C 180,E1 -5680.259,E2 -5680.259} C_VEL
LIN {X 0,Y 503.496,Z 549.353,A -85,B 0,C 180,E1 -5681.269,E2 -5681.269} C_VEL
LIN {X 0,Y 503.874,Z 539.702,A -85,B 0,C 180,E1 -5682.076,E2 -5682.076} C_VEL
LIN {X 0,Y 504.156,Z 528.732,A -85,B 0,C 180,E1 -5682.817,E2 -5682.817} C_VEL
LIN {X 0,Y 504.478,Z 516.701,A -85,B 0,C 180,E1 -5683.443,E2 -5683.443} C_VEL
LIN {X 0,Y 504.779,Z 503.364,A -85,B 0,C 180,E1 -5683.948,E2 -5683.948} C_VEL
LIN {X 0,Y 504.938,Z 490.89,A -85,B 0,C 180,E1 -5684.251,E2 -5684.251} C_VEL
LIN {X 0,Y 505.39,Z 396.906,A -85,B 0,C 180,E1 -5685.605,E2 -5685.605} C_VEL
LIN {X 0,Y 503.298,Z 385.98,A -85,B 0,C 180,E1 -5685.848,E2 -5685.848} C_VEL
LIN {X 0,Y 503.792,Z 370.003,A -85,B 0,C 180,E1 -5689.137,E2 -5689.137} C_VEL
LIN {X 0,Y 502.861,Z 363.851,A -85,B 0,C 180,E1 -5690.49,E2 -5690.49} C_VEL
LIN {X 0,Y 502.794,Z 363.86,A -85,B 0,C 180,E1 -5693.913,E2 -5693.913} C_VEL
LIN {X 0,Y 502.865,Z 363.843,A -85,B 0,C 180,E1 -5696.565,E2 -5696.565} C_VEL
LIN {X 0,Y 502.824,Z 363.847,A -85,B 0,C 180,E1 -5699.287,E2 -5699.287} C_VEL
LIN {X 0,Y 502.785,Z 363.857,A -85,B 0,C 180,E1 -5702.084,E2 -5702.084} C_VEL
LIN {X 0,Y 502.809,Z 363.848,A -85,B 0,C 180,E1 -5704.964,E2 -5704.964} C_VEL
LIN {X 0,Y 502.792,Z 363.857,A -85,B 0,C 180,E1 -5707.953,E2 -5707.953} C_VEL
LIN {X 0,Y 502.817,Z 363.847,A -85,B 0,C 180,E1 -5711.065,E2 -5711.065} C_VEL
LIN {X 0,Y 502.797,Z 363.85,A -85,B 0,C 180,E1 -5714.531,E2 -5714.531} C_VEL
LIN {X 0,Y 502.831,Z 363.852,A -85,B 0,C 180,E1 -5717.864,E2 -5717.864} C_VEL
LIN {X 0,Y 502.805,Z 363.85,A -85,B 0,C 180,E1 -5721.024,E2 -5721.024} C_VEL
LIN {X 0,Y 502.78,Z 363.853,A -85,B 0,C 180,E1 -5724.166,E2 -5724.166} C_VEL
LIN {X 0,Y 502.827,Z 363.847,A -85,B 0,C 180,E1 -5726.992,E2 -5726.992} C_VEL
LIN {X 0,Y 502.808,Z 363.85,A -85,B 0,C 180,E1 -5730.064,E2 -5730.064} C_VEL
LIN {X 0,Y 502.828,Z 363.845,A -85,B 0,C 180,E1 -5732.533,E2 -5732.533} C_VEL
LIN {X 0,Y 502.823,Z 363.853,A -85,B 0,C 180,E1 -5735.297,E2 -5735.297} C_VEL
LIN {X 0,Y 502.803,Z 363.852,A -85,B 0,C 180,E1 -5737.827,E2 -5737.827} C_VEL
LIN {X 0,Y 502.818,Z 363.847,A -85,B 0,C 180,E1 -5740.4,E2 -5740.4} C_VEL
LIN {X 0,Y 502.828,Z 363.849,A -85,B 0,C 180,E1 -5742.931,E2 -5742.931} C_VEL
LIN {X 0,Y 502.843,Z 363.851,A -85,B 0,C 180,E1 -5745.429,E2 -5745.429} C_VEL
LIN {X 0,Y 502.886,Z 363.84,A -85,B 0,C 180,E1 -5748.717,E2 -5748.717} C_VEL
LIN {X 0,Y 502.893,Z 363.838,A -85,B 0,C 180,E1 -5751.966,E2 -5751.966} C_VEL
LIN {X 0,Y 502.931,Z 363.833,A -85,B 0,C 180,E1 -5754.386,E2 -5754.386} C_VEL
LIN {X 0,Y 503.017,Z 363.825,A -85,B 0,C 180,E1 -5757.598,E2 -5757.598} C_VEL
LIN {X 0,Y 503.017,Z 363.822,A -85,B 0,C 180,E1 -5760,E2 -5760} C_VEL
LIN {X 0,Y 503.017,Z 363.823,A -85,B 0,C 180,E1 -5762.402,E2 -5762.402} C_VEL
LIN {X 0,Y 502.94,Z 363.833,A -85,B 0,C 180,E1 -5765.613,E2 -5765.613} C_VEL
LIN {X 0,Y 502.894,Z 363.837,A -85,B 0,C 180,E1 -5768.033,E2 -5768.033} C_VEL
LIN {X 0,Y 502.889,Z 363.842,A -85,B 0,C 180,E1 -5771.283,E2 -5771.283} C_VEL
LIN {X 0,Y 502.836,Z 363.849,A -85,B 0,C 180,E1 -5774.571,E2 -5774.571} C_VEL
LIN {X 0,Y 502.853,Z 363.842,A -85,B 0,C 180,E1 -5777.907,E2 -5777.907} C_VEL
LIN {X 0,Y 502.822,Z 363.851,A -85,B 0,C 180,E1 -5780.537,E2 -5780.537} C_VEL
LIN {X 0,Y 502.798,Z 363.854,A -85,B 0,C 180,E1 -5783.04,E2 -5783.04} C_VEL
LIN {X 0,Y 502.835,Z 363.845,A -85,B 0,C 180,E1 -5785.676,E2 -5785.676} C_VEL
LIN {X 0,Y 502.833,Z 363.849,A -85,B 0,C 180,E1 -5788.373,E2 -5788.373} C_VEL
LIN {X 0,Y 502.789,Z 363.85,A -85,B 0,C 180,E1 -5791.5,E2 -5791.5} C_VEL
LIN {X 0,Y 502.801,Z 363.855,A -85,B 0,C 180,E1 -5794.446,E2 -5794.446} C_VEL
LIN {X 0,Y 502.775,Z 363.853,A -85,B 0,C 180,E1 -5797.179,E2 -5797.179} C_VEL
LIN {X 0,Y 502.817,Z 363.849,A -85,B 0,C 180,E1 -5800.013,E2 -5800.013} C_VEL
LIN {X 0,Y 502.825,Z 363.85,A -85,B 0,C 180,E1 -5802.203,E2 -5802.203} C_VEL
LIN {X 0,Y 502.797,Z 363.849,A -85,B 0,C 180,E1 -5805.469,E2 -5805.469} C_VEL
LIN {X 0,Y 502.826,Z 363.847,A -85,B 0,C 180,E1 -5807.865,E2 -5807.865} C_VEL
LIN {X 0,Y 502.8,Z 363.85,A -85,B 0,C 180,E1 -5811.025,E2 -5811.025} C_VEL
LIN {X 0,Y 502.784,Z 363.857,A -85,B 0,C 180,E1 -5814.168,E2 -5814.168} C_VEL
LIN {X 0,Y 502.832,Z 363.846,A -85,B 0,C 180,E1 -5816.994,E2 -5816.994} C_VEL
LIN {X 0,Y 502.814,Z 363.853,A -85,B 0,C 180,E1 -5820.066,E2 -5820.066} C_VEL
LIN {X 0,Y 502.834,Z 363.852,A -85,B 0,C 180,E1 -5822.534,E2 -5822.534} C_VEL
LIN {X 0,Y 502.861,Z 363.939,A -85,B 0,C 180,E1 -5824.825,E2 -5824.825} C_VEL
LIN {X 0,Y 504.657,Z 373.75,A -85,B 0,C 180,E1 -5826.552,E2 -5826.552} C_VEL
LIN {X 0,Y 504.145,Z 390.78,A -85,B 0,C 180,E1 -5829.329,E2 -5829.329} C_VEL
LIN {X 0,Y 503.555,Z 410.747,A -85,B 0,C 180,E1 -5832.539,E2 -5832.539} C_VEL
LIN {X 0,Y 503.307,Z 421.115,A -85,B 0,C 180,E1 -5834.194,E2 -5834.194} C_VEL
LIN {X 0,Y 505.379,Z 434.951,A -85,B 0,C 180,E1 -5834.46,E2 -5834.46} C_VEL
LIN {X 0,Y 504.861,Z 529.437,A -85,B 0,C 180,E1 -5835.823,E2 -5835.823} C_VEL
LIN {X 0,Y 504.575,Z 542.721,A -85,B 0,C 180,E1 -5836.175,E2 -5836.175} C_VEL
LIN {X 0,Y 504.235,Z 556.021,A -85,B 0,C 180,E1 -5836.705,E2 -5836.705} C_VEL
LIN {X 0,Y 503.842,Z 568.504,A -85,B 0,C 180,E1 -5837.394,E2 -5837.394} C_VEL
LIN {X 0,Y 503.533,Z 580.099,A -85,B 0,C 180,E1 -5838.222,E2 -5838.222} C_VEL
LIN {X 0,Y 503.204,Z 590.309,A -85,B 0,C 180,E1 -5839.132,E2 -5839.132} C_VEL
LIN {X 0,Y 502.849,Z 599.496,A -85,B 0,C 180,E1 -5840.142,E2 -5840.142} C_VEL
LIN {X 0,Y 502.578,Z 608.453,A -85,B 0,C 180,E1 -5841.354,E2 -5841.354} C_VEL
LIN {X 0,Y 502.349,Z 615.662,A -85,B 0,C 180,E1 -5842.565,E2 -5842.565} C_VEL
LIN {X 0,Y 502.235,Z 620.529,A -85,B 0,C 180,E1 -5843.573,E2 -5843.573} C_VEL
LIN {X 0,Y 502.175,Z 625.262,A -85,B 0,C 180,E1 -5844.781,E2 -5844.781} C_VEL
LIN {X 0,Y 502.139,Z 628.877,A -85,B 0,C 180,E1 -5845.987,E2 -5845.987} C_VEL
LIN {X 0,Y 502.12,Z 630.742,A -85,B 0,C 180,E1 -5846.791,E2 -5846.791} C_VEL
LIN {X 0,Y 502.091,Z 632.14,A -85,B 0,C 180,E1 -5847.593,E2 -5847.593} C_VEL
LIN {X 0,Y 501.99,Z 633.744,A -85,B 0,C 180,E1 -5849.198,E2 -5849.198} C_VEL
LIN {X 0,Y 501.981,Z 633.961,A -85,B 0,C 180,E1 -5850,E2 -5850} C_VEL
LIN {X 0,Y 502.036,Z 633.138,A -85,B 0,C 180,E1 -5851.604,E2 -5851.604} C_VEL
LIN {X 0,Y 502.091,Z 632.143,A -85,B 0,C 180,E1 -5852.407,E2 -5852.407} C_VEL
LIN {X 0,Y 502.12,Z 630.746,A -85,B 0,C 180,E1 -5853.209,E2 -5853.209} C_VEL
LIN {X 0,Y 502.103,Z 627.804,A -85,B 0,C 180,E1 -5854.415,E2 -5854.415} C_VEL
LIN {X 0,Y 502.211,Z 623.826,A -85,B 0,C 180,E1 -5855.622,E2 -5855.622} C_VEL
LIN {X 0,Y 502.333,Z 617.807,A -85,B 0,C 180,E1 -5857.011,E2 -5857.011} C_VEL
LIN {X 0,Y 502.482,Z 611.017,A -85,B 0,C 180,E1 -5858.242,E2 -5858.242} C_VEL
LIN {X 0,Y 502.724,Z 602.721,A -85,B 0,C 180,E1 -5859.454,E2 -5859.454} C_VEL
LIN {X 0,Y 503.001,Z 594.221,A -85,B 0,C 180,E1 -5860.465,E2 -5860.465} C_VEL
LIN {X 0,Y 503.414,Z 583.722,A -85,B 0,C 180,E1 -5861.475,E2 -5861.475} C_VEL
LIN {X 0,Y 503.683,Z 573.407,A -85,B 0,C 180,E1 -5862.28,E2 -5862.28} C_VEL
LIN {X 0,Y 504.115,Z 561.954,A -85,B 0,C 180,E1 -5862.991,E2 -5862.991} C_VEL
LIN {X 0,Y 504.412,Z 550.284,A -85,B 0,C 180,E1 -5863.547,E2 -5863.547} C_VEL
LIN {X 0,Y 504.694,Z 536.84,A -85,B 0,C 180,E1 -5864.001,E2 -5864.001} C_VEL
LIN {X 0,Y 504.961,Z 523.576,A -85,B 0,C 180,E1 -5864.277,E2 -5864.277} C_VEL
LIN {X 0,Y 505.236,Z 433.85,A -85,B 0,C 180,E1 -5865.56,E2 -5865.56} C_VEL
LIN {X 0,Y 503.308,Z 421.003,A -85,B 0,C 180,E1 -5865.825,E2 -5865.825} C_VEL
LIN {X 0,Y 503.868,Z 400.315,A -85,B 0,C 180,E1 -5869.134,E2 -5869.134} C_VEL
LIN {X 0,Y 504.502,Z 380.689,A -85,B 0,C 180,E1 -5872.309,E2 -5872.309} C_VEL
LIN {X 0,Y 504.662,Z 373.712,A -85,B 0,C 180,E1 -5873.454,E2 -5873.454} C_VEL
LIN {X 0,Y 502.852,Z 363.851,A -85,B 0,C 180,E1 -5875.23,E2 -5875.23} C_VEL
LIN {X 0,Y 502.844,Z 363.849,A -85,B 0,C 180,E1 -5878.295,E2 -5878.295} C_VEL
LIN {X 0,Y 502.796,Z 363.858,A -85,B 0,C 180,E1 -5881.499,E2 -5881.499} C_VEL
LIN {X 0,Y 502.805,Z 363.849,A -85,B 0,C 180,E1 -5884.444,E2 -5884.444} C_VEL
LIN {X 0,Y 502.779,Z 363.854,A -85,B 0,C 180,E1 -5887.178,E2 -5887.178} C_VEL
LIN {X 0,Y 502.786,Z 363.854,A -85,B 0,C 180,E1 -5890.014,E2 -5890.014} C_VEL
LIN {X 0,Y 502.799,Z 363.85,A -85,B 0,C 180,E1 -5892.198,E2 -5892.198} C_VEL
LIN {X 0,Y 502.797,Z 363.857,A -85,B 0,C 180,E1 -5895.467,E2 -5895.467} C_VEL
LIN {X 0,Y 502.831,Z 363.849,A -85,B 0,C 180,E1 -5897.864,E2 -5897.864} C_VEL
LIN {X 0,Y 502.805,Z 363.851,A -85,B 0,C 180,E1 -5901.024,E2 -5901.024} C_VEL
LIN {X 0,Y 502.78,Z 363.852,A -85,B 0,C 180,E1 -5904.166,E2 -5904.166} C_VEL
LIN {X 0,Y 502.826,Z 363.849,A -85,B 0,C 180,E1 -5906.992,E2 -5906.992} C_VEL
LIN {X 0,Y 502.824,Z 363.847,A -85,B 0,C 180,E1 -5910.061,E2 -5910.061} C_VEL
LIN {X 0,Y 502.828,Z 363.846,A -85,B 0,C 180,E1 -5912.533,E2 -5912.533} C_VEL
LIN {X 0,Y 502.823,Z 363.855,A -85,B 0,C 180,E1 -5915.297,E2 -5915.297} C_VEL
LIN {X 0,Y 502.803,Z 363.85,A -85,B 0,C 180,E1 -5917.827,E2 -5917.827} C_VEL
LIN {X 0,Y 502.818,Z 363.847,A -85,B 0,C 180,E1 -5920.4,E2 -5920.4} C_VEL
LIN {X 0,Y 502.828,Z 363.851,A -85,B 0,C 180,E1 -5922.931,E2 -5922.931} C_VEL
LIN {X 0,Y 502.836,Z 363.849,A -85,B 0,C 180,E1 -5925.429,E2 -5925.429} C_VEL
LIN {X 0,Y 502.888,Z 363.842,A -85,B 0,C 180,E1 -5928.717,E2 -5928.717} C_VEL
LIN {X 0,Y 502.893,Z 363.837,A -85,B 0,C 180,E1 -5931.967,E2 -5931.967} C_VEL
LIN {X 0,Y 502.931,Z 363.834,A -85,B 0,C 180,E1 -5934.386,E2 -5934.386} C_VEL
LIN {X 0,Y 503.017,Z 363.823,A -85,B 0,C 180,E1 -5937.598,E2 -5937.598} C_VEL
LIN {X 0,Y 503.017,Z 363.822,A -85,B 0,C 180,E1 -5940,E2 -5940} C_VEL
LIN {X 0,Y 503.017,Z 363.824,A -85,B 0,C 180,E1 -5942.402,E2 -5942.402} C_VEL
LIN {X 0,Y 502.94,Z 363.832,A -85,B 0,C 180,E1 -5945.614,E2 -5945.614} C_VEL
LIN {X 0,Y 502.893,Z 363.838,A -85,B 0,C 180,E1 -5948.034,E2 -5948.034} C_VEL
LIN {X 0,Y 502.886,Z 363.841,A -85,B 0,C 180,E1 -5951.283,E2 -5951.283} C_VEL
LIN {X 0,Y 502.843,Z 363.85,A -85,B 0,C 180,E1 -5954.571,E2 -5954.571} C_VEL
LIN {X 0,Y 502.853,Z 363.843,A -85,B 0,C 180,E1 -5957.907,E2 -5957.907} C_VEL
LIN {X 0,Y 502.822,Z 363.853,A -85,B 0,C 180,E1 -5960.537,E2 -5960.537} C_VEL
LIN {X 0,Y 502.798,Z 363.852,A -85,B 0,C 180,E1 -5963.04,E2 -5963.04} C_VEL
LIN {X 0,Y 502.835,Z 363.845,A -85,B 0,C 180,E1 -5965.676,E2 -5965.676} C_VEL
LIN {X 0,Y 502.834,Z 363.851,A -85,B 0,C 180,E1 -5968.373,E2 -5968.373} C_VEL
LIN {X 0,Y 502.789,Z 363.85,A -85,B 0,C 180,E1 -5971.5,E2 -5971.5} C_VEL
LIN {X 0,Y 502.798,Z 363.858,A -85,B 0,C 180,E1 -5974.445,E2 -5974.445} C_VEL
LIN {X 0,Y 502.776,Z 363.853,A -85,B 0,C 180,E1 -5977.179,E2 -5977.179} C_VEL
LIN {X 0,Y 502.817,Z 363.85,A -85,B 0,C 180,E1 -5980.013,E2 -5980.013} C_VEL
LIN {X 0,Y 502.819,Z 363.853,A -85,B 0,C 180,E1 -5982.203,E2 -5982.203} C_VEL
LIN {X 0,Y 502.797,Z 363.85,A -85,B 0,C 180,E1 -5985.469,E2 -5985.469} C_VEL
LIN {X 0,Y 502.817,Z 363.848,A -85,B 0,C 180,E1 -5988.935,E2 -5988.935} C_VEL
LIN {X 0,Y 502.792,Z 363.856,A -85,B 0,C 180,E1 -5992.047,E2 -5992.047} C_VEL
LIN {X 0,Y 502.809,Z 363.848,A -85,B 0,C 180,E1 -5995.036,E2 -5995.036} C_VEL
LIN {X 0,Y 502.806,Z 363.848,A -85,B 0,C 180,E1 -5997.242,E2 -5997.242} C_VEL
LIN {X 0,Y 502.106,Z 363.943,A -85,B 0,C 180,E1 -5997.911,E2 -5997.911} C_VEL
LIN {X 0,Y 499.242,Z 364.297,A -85,B 0,C 180,E1 -5998.997,E2 -5998.997} C_VEL
LIN {X 0,Y 496.848,Z 364.596,A -85,B 0,C 180,E1 -5999.872,E2 -5999.872} C_VEL
LIN {X 0,Y 495.832,Z 364.721,A -85,B 0,C 180,E1 -6000.547,E2 -6000.547} C_VEL
LIN {X 0,Y 495.755,Z 364.728,A -85,B 0,C 180,E1 -6000.776,E2 -6000.776} C_VEL
LIN {X 0,Y 495.824,Z 364.718,A -85,B 0,C 180,E1 -6003.251,E2 -6003.251} C_VEL
LIN {X 0,Y 495.744,Z 364.733,A -85,B 0,C 180,E1 -6006.613,E2 -6006.613} C_VEL
LIN {X 0,Y 495.815,Z 364.911,A -85,B 0,C 180,E1 -6009.49,E2 -6009.49} C_VEL
LIN {X 0,Y 496.783,Z 370.79,A -85,B 0,C 180,E1 -6010.797,E2 -6010.797} C_VEL
LIN {X 0,Y 496.359,Z 383.962,A -85,B 0,C 180,E1 -6013.55,E2 -6013.55} C_VEL
LIN {X 0,Y 496.325,Z 386.348,A -85,B 0,C 180,E1 -6014.032,E2 -6014.032} C_VEL
LIN {X 0,Y 498.673,Z 398.893,A -85,B 0,C 180,E1 -6014.295,E2 -6014.295} C_VEL
LIN {X 0,Y 498.064,Z 493.173,A -85,B 0,C 180,E1 -6015.678,E2 -6015.678} C_VEL
LIN {X 0,Y 497.803,Z 506.307,A -85,B 0,C 180,E1 -6016.035,E2 -6016.035} C_VEL
LIN {X 0,Y 497.524,Z 519.486,A -85,B 0,C 180,E1 -6016.574,E2 -6016.574} C_VEL
LIN {X 0,Y 497.217,Z 531.301,A -85,B 0,C 180,E1 -6017.238,E2 -6017.238} C_VEL
LIN {X 0,Y 496.841,Z 542.701,A -85,B 0,C 180,E1 -6018.061,E2 -6018.061} C_VEL
LIN {X 0,Y 496.403,Z 552.938,A -85,B 0,C 180,E1 -6018.981,E2 -6018.981} C_VEL
LIN {X 0,Y 496.079,Z 562.118,A -85,B 0,C 180,E1 -6020.006,E2 -6020.006} C_VEL
LIN {X 0,Y 495.721,Z 571.026,A -85,B 0,C 180,E1 -6021.234,E2 -6021.234} C_VEL
LIN {X 0,Y 495.449,Z 578.197,A -85,B 0,C 180,E1 -6022.461,E2 -6022.461} C_VEL
LIN {X 0,Y 495.298,Z 583.034,A -85,B 0,C 180,E1 -6023.482,E2 -6023.482} C_VEL
LIN {X 0,Y 495.129,Z 587.735,A -85,B 0,C 180,E1 -6024.706,E2 -6024.706} C_VEL
LIN {X 0,Y 495.172,Z 591.328,A -85,B 0,C 180,E1 -6025.931,E2 -6025.931} C_VEL
LIN {X 0,Y 495.051,Z 593.192,A -85,B 0,C 180,E1 -6026.745,E2 -6026.745} C_VEL
LIN {X 0,Y 495.054,Z 594.593,A -85,B 0,C 180,E1 -6027.559,E2 -6027.559} C_VEL
LIN {X 0,Y 494.911,Z 596.209,A -85,B 0,C 180,E1 -6029.186,E2 -6029.186} C_VEL
LIN {X 0,Y 494.901,Z 596.446,A -85,B 0,C 180,E1 -6030,E2 -6030} C_VEL
LIN {X 0,Y 494.911,Z 596.261,A -85,B 0,C 180,E1 -6030.814,E2 -6030.814} C_VEL
LIN {X 0,Y 495.054,Z 594.713,A -85,B 0,C 180,E1 -6032.441,E2 -6032.441} C_VEL
LIN {X 0,Y 495.051,Z 593.364,A -85,B 0,C 180,E1 -6033.255,E2 -6033.255} C_VEL
LIN {X 0,Y 495.141,Z 590.506,A -85,B 0,C 180,E1 -6034.477,E2 -6034.477} C_VEL
LIN {X 0,Y 495.242,Z 586.632,A -85,B 0,C 180,E1 -6035.701,E2 -6035.701} C_VEL
LIN {X 0,Y 495.363,Z 581.635,A -85,B 0,C 180,E1 -6036.926,E2 -6036.926} C_VEL
LIN {X 0,Y 495.531,Z 575.343,A -85,B 0,C 180,E1 -6038.153,E2 -6038.153} C_VEL
LIN {X 0,Y 495.818,Z 567.461,A -85,B 0,C 180,E1 -6039.381,E2 -6039.381} C_VEL
LIN {X 0,Y 496.138,Z 559.424,A -85,B 0,C 180,E1 -6040.405,E2 -6040.405} C_VEL
LIN {X 0,Y 496.545,Z 549.613,A -85,B 0,C 180,E1 -6041.429,E2 -6041.429} C_VEL
LIN {X 0,Y 496.987,Z 538.506,A -85,B 0,C 180,E1 -6042.356,E2 -6042.356} C_VEL
LIN {X 0,Y 497.309,Z 527.77,A -85,B 0,C 180,E1 -6043.068,E2 -6043.068} C_VEL
LIN {X 0,Y 497.607,Z 515.827,A -85,B 0,C 180,E1 -6043.684,E2 -6043.684} C_VEL
LIN {X 0,Y 497.909,Z 502.747,A -85,B 0,C 180,E1 -6044.17,E2 -6044.17} C_VEL
LIN {X 0,Y 498.092,Z 489.615,A -85,B 0,C 180,E1 -6044.478,E2 -6044.478} C_VEL
LIN {X 0,Y 498.543,Z 397.569,A -85,B 0,C 180,E1 -6045.818,E2 -6045.818} C_VEL
LIN {X 0,Y 496.308,Z 386.31,A -85,B 0,C 180,E1 -6046.059,E2 -6046.059} C_VEL
LIN {X 0,Y 496.823,Z 371.227,A -85,B 0,C 180,E1 -6049.201,E2 -6049.201} C_VEL
LIN {X 0,Y 495.78,Z 364.732,A -85,B 0,C 180,E1 -6050.675,E2 -6050.675} C_VEL
LIN {X 0,Y 495.755,Z 364.734,A -85,B 0,C 180,E1 -6053.386,E2 -6053.386} C_VEL
LIN {X 0,Y 495.792,Z 364.73,A -85,B 0,C 180,E1 -6056.067,E2 -6056.067} C_VEL
LIN {X 0,Y 495.772,Z 364.725,A -85,B 0,C 180,E1 -6058.814,E2 -6058.814} C_VEL
LIN {X 0,Y 495.756,Z 364.732,A -85,B 0,C 180,E1 -6061.725,E2 -6061.725} C_VEL
LIN {X 0,Y 495.776,Z 364.724,A -85,B 0,C 180,E1 -6064.695,E2 -6064.695} C_VEL
LIN {X 0,Y 495.73,Z 364.734,A -85,B 0,C 180,E1 -6067.561,E2 -6067.561} C_VEL
LIN {X 0,Y 495.764,Z 364.726,A -85,B 0,C 180,E1 -6070.699,E2 -6070.699} C_VEL
LIN {X 0,Y 495.73,Z 364.735,A -85,B 0,C 180,E1 -6074,E2 -6074} C_VEL
LIN {X 0,Y 495.758,Z 364.728,A -85,B 0,C 180,E1 -6077.12,E2 -6077.12} C_VEL
LIN {X 0,Y 495.778,Z 364.725,A -85,B 0,C 180,E1 -6080.364,E2 -6080.364} C_VEL
LIN {X 0,Y 495.729,Z 364.736,A -85,B 0,C 180,E1 -6083.456,E2 -6083.456} C_VEL
LIN {X 0,Y 495.755,Z 364.727,A -85,B 0,C 180,E1 -6086.435,E2 -6086.435} C_VEL
LIN {X 0,Y 495.745,Z 364.733,A -85,B 0,C 180,E1 -6089.312,E2 -6089.312} C_VEL
LIN {X 0,Y 495.775,Z 364.725,A -85,B 0,C 180,E1 -6092.108,E2 -6092.108} C_VEL
LIN {X 0,Y 495.783,Z 364.724,A -85,B 0,C 180,E1 -6094.832,E2 -6094.832} C_VEL
LIN {X 0,Y 495.753,Z 364.735,A -85,B 0,C 180,E1 -6097.495,E2 -6097.495} C_VEL
LIN {X 0,Y 495.77,Z 364.725,A -85,B 0,C 180,E1 -6100.109,E2 -6100.109} C_VEL
LIN {X 0,Y 495.78,Z 364.724,A -85,B 0,C 180,E1 -6102.681,E2 -6102.681} C_VEL
LIN {X 0,Y 495.786,Z 364.73,A -85,B 0,C 180,E1 -6105.217,E2 -6105.217} C_VEL
LIN {X 0,Y 495.86,Z 364.714,A -85,B 0,C 180,E1 -6108.555,E2 -6108.555} C_VEL
LIN {X 0,Y 495.865,Z 364.714,A -85,B 0,C 180,E1 -6111.852,E2 -6111.852} C_VEL
LIN {X 0,Y 495.888,Z 364.71,A -85,B 0,C 180,E1 -6114.306,E2 -6114.306} C_VEL
LIN {X 0,Y 495.986,Z 364.701,A -85,B 0,C 180,E1 -6117.564,E2 -6117.564} C_VEL
LIN {X 0,Y 495.988,Z 364.698,A -85,B 0,C 180,E1 -6120,E2 -6120} C_VEL
LIN {X 0,Y 495.986,Z 364.699,A -85,B 0,C 180,E1 -6122.436,E2 -6122.436} C_VEL
LIN {X 0,Y 495.896,Z 364.71,A -85,B 0,C 180,E1 -6125.693,E2 -6125.693} C_VEL
LIN {X 0,Y 495.865,Z 364.713,A -85,B 0,C 180,E1 -6128.148,E2 -6128.148} C_VEL
LIN {X 0,Y 495.868,Z 364.715,A -85,B 0,C 180,E1 -6131.445,E2 -6131.445} C_VEL
LIN {X 0,Y 495.781,Z 364.731,A -85,B 0,C 180,E1 -6134.783,E2 -6134.783} C_VEL
LIN {X 0,Y 495.78,Z 364.726,A -85,B 0,C 180,E1 -6137.319,E2 -6137.319} C_VEL
LIN {X 0,Y 495.77,Z 364.725,A -85,B 0,C 180,E1 -6139.89,E2 -6139.89} C_VEL
LIN {X 0,Y 495.757,Z 364.734,A -85,B 0,C 180,E1 -6142.863,E2 -6142.863} C_VEL
LIN {X 0,Y 495.792,Z 364.723,A -85,B 0,C 180,E1 -6146.068,E2 -6146.068} C_VEL
LIN {X 0,Y 495.766,Z 364.732,A -85,B 0,C 180,E1 -6148.815,E2 -6148.815} C_VEL
LIN {X 0,Y 495.752,Z 364.727,A -85,B 0,C 180,E1 -6151.727,E2 -6151.727} C_VEL
LIN {X 0,Y 495.771,Z 364.732,A -85,B 0,C 180,E1 -6154.696,E2 -6154.696} C_VEL
LIN {X 0,Y 495.726,Z 364.73,A -85,B 0,C 180,E1 -6157.562,E2 -6157.562} C_VEL
LIN {X 0,Y 495.775,Z 364.73,A -85,B 0,C 180,E1 -6160.699,E2 -6160.699} C_VEL
LIN {X 0,Y 495.73,Z 364.73,A -85,B 0,C 180,E1 -6163.696,E2 -6163.696} C_VEL
LIN {X 0,Y 495.731,Z 364.736,A -85,B 0,C 180,E1 -6166.305,E2 -6166.305} C_VEL
LIN {X 0,Y 495.764,Z 364.726,A -85,B 0,C 180,E1 -6169.301,E2 -6169.301} C_VEL
LIN {X 0,Y 495.73,Z 364.737,A -85,B 0,C 180,E1 -6172.439,E2 -6172.439} C_VEL
LIN {X 0,Y 495.784,Z 364.723,A -85,B 0,C 180,E1 -6175.458,E2 -6175.458} C_VEL
LIN {X 0,Y 495.759,Z 364.735,A -85,B 0,C 180,E1 -6178.365,E2 -6178.365} C_VEL
LIN {X 0,Y 495.788,Z 364.726,A -85,B 0,C 180,E1 -6181.507,E2 -6181.507} C_VEL
LIN {X 0,Y 495.825,Z 364.726,A -85,B 0,C 180,E1 -6184.611,E2 -6184.611} C_VEL
LIN {X 0,Y 497.58,Z 373.908,A -85,B 0,C 180,E1 -6186.264,E2 -6186.264} C_VEL
LIN {X 0,Y 497.572,Z 381.771,A -85,B 0,C 180,E1 -6187.582,E2 -6187.582} C_VEL
LIN {X 0,Y 496.859,Z 401.391,A -85,B 0,C 180,E1 -6190.8,E2 -6190.8} C_VEL
LIN {X 0,Y 496.271,Z 420.836,A -85,B 0,C 180,E1 -6193.963,E2 -6193.963} C_VEL
LIN {X 0,Y 498.533,Z 435.858,A -85,B 0,C 180,E1 -6194.258,E2 -6194.258} C_VEL
LIN {X 0,Y 497.999,Z 529.17,A -85,B 0,C 180,E1 -6195.624,E2 -6195.624} C_VEL
LIN {X 0,Y 497.665,Z 542.453,A -85,B 0,C 180,E1 -6195.979,E2 -6195.979} C_VEL
LIN {X 0,Y 497.318,Z 555.754,A -85,B 0,C 180,E1 -6196.516,E2 -6196.516} C_VEL
LIN {X 0,Y 496.9,Z 568.243,A -85,B 0,C 180,E1 -6197.216,E2 -6197.216} C_VEL
LIN {X 0,Y 496.541,Z 579.83,A -85,B 0,C 180,E1 -6198.054,E2 -6198.054} C_VEL
LIN {X 0,Y 496.207,Z 590.041,A -85,B 0,C 180,E1 -6198.977,E2 -6198.977} C_VEL
LIN {X 0,Y 495.818,Z 599.228,A -85,B 0,C 180,E1 -6200.001,E2 -6200.001} C_VEL
LIN {X 0,Y 495.503,Z 608.184,A -85,B 0,C 180,E1 -6201.23,E2 -6201.23} C_VEL
LIN {X 0,Y 495.281,Z 615.394,A -85,B 0,C 180,E1 -6202.458,E2 -6202.458} C_VEL
LIN {X 0,Y 495.126,Z 621.438,A -85,B 0,C 180,E1 -6203.757,E2 -6203.757} C_VEL
LIN {X 0,Y 495.037,Z 626.307,A -85,B 0,C 180,E1 -6205.114,E2 -6205.114} C_VEL
LIN {X 0,Y 495.033,Z 628.609,A -85,B 0,C 180,E1 -6205.93,E2 -6205.93} C_VEL
LIN {X 0,Y 495.042,Z 630.476,A -85,B 0,C 180,E1 -6206.745,E2 -6206.745} C_VEL
LIN {X 0,Y 494.998,Z 631.873,A -85,B 0,C 180,E1 -6207.559,E2 -6207.559} C_VEL
LIN {X 0,Y 494.962,Z 632.87,A -85,B 0,C 180,E1 -6208.373,E2 -6208.373} C_VEL
LIN {X 0,Y 494.898,Z 633.694,A -85,B 0,C 180,E1 -6210,E2 -6210} C_VEL
LIN {X 0,Y 494.962,Z 632.872,A -85,B 0,C 180,E1 -6211.627,E2 -6211.627} C_VEL
LIN {X 0,Y 494.998,Z 631.876,A -85,B 0,C 180,E1 -6212.441,E2 -6212.441} C_VEL
LIN {X 0,Y 495.042,Z 630.479,A -85,B 0,C 180,E1 -6213.255,E2 -6213.255} C_VEL
LIN {X 0,Y 495.009,Z 627.536,A -85,B 0,C 180,E1 -6214.479,E2 -6214.479} C_VEL
LIN {X 0,Y 495.128,Z 623.558,A -85,B 0,C 180,E1 -6215.702,E2 -6215.702} C_VEL
LIN {X 0,Y 495.256,Z 617.437,A -85,B 0,C 180,E1 -6217.133,E2 -6217.133} C_VEL
LIN {X 0,Y 495.429,Z 610.749,A -85,B 0,C 180,E1 -6218.36,E2 -6218.36} C_VEL
LIN {X 0,Y 495.686,Z 602.453,A -85,B 0,C 180,E1 -6219.59,E2 -6219.59} C_VEL
LIN {X 0,Y 495.995,Z 593.953,A -85,B 0,C 180,E1 -6220.614,E2 -6220.614} C_VEL
LIN {X 0,Y 496.432,Z 583.454,A -85,B 0,C 180,E1 -6221.638,E2 -6221.638} C_VEL
LIN {X 0,Y 496.754,Z 572.176,A -85,B 0,C 180,E1 -6222.524,E2 -6222.524} C_VEL
LIN {X 0,Y 497.159,Z 561.686,A -85,B 0,C 180,E1 -6223.176,E2 -6223.176} C_VEL
LIN {X 0,Y 497.48,Z 550.015,A -85,B 0,C 180,E1 -6223.74,E2 -6223.74} C_VEL
LIN {X 0,Y 497.793,Z 537.489,A -85,B 0,C 180,E1 -6224.173,E2 -6224.173} C_VEL
LIN {X 0,Y 498.047,Z 524.823,A -85,B 0,C 180,E1 -6224.453,E2 -6224.453} C_VEL
LIN {X 0,Y 498.467,Z 435.149,A -85,B 0,C 180,E1 -6225.754,E2 -6225.754} C_VEL
LIN {X 0,Y 496.282,Z 420.848,A -85,B 0,C 180,E1 -6226.036,E2 -6226.036} C_VEL
LIN {X 0,Y 496.865,Z 401.378,A -85,B 0,C 180,E1 -6229.199,E2 -6229.199} C_VEL
LIN {X 0,Y 497.575,Z 381.767,A -85,B 0,C 180,E1 -6232.417,E2 -6232.417} C_VEL
LIN {X 0,Y 497.746,Z 375.878,A -85,B 0,C 180,E1 -6233.396,E2 -6233.396} C_VEL
LIN {X 0,Y 496.255,Z 366.883,A -85,B 0,C 180,E1 -6234.991,E2 -6234.991} C_VEL
LIN {X 0,Y 495.825,Z 364.726,A -85,B 0,C 180,E1 -6235.389,E2 -6235.389} C_VEL
LIN {X 0,Y 495.788,Z 364.726,A -85,B 0,C 180,E1 -6238.493,E2 -6238.493} C_VEL
LIN {X 0,Y 495.758,Z 364.735,A -85,B 0,C 180,E1 -6241.725,E2 -6241.725} C_VEL
LIN {X 0,Y 495.775,Z 364.724,A -85,B 0,C 180,E1 -6244.695,E2 -6244.695} C_VEL
LIN {X 0,Y 495.73,Z 364.737,A -85,B 0,C 180,E1 -6247.561,E2 -6247.561} C_VEL
LIN {X 0,Y 495.764,Z 364.726,A -85,B 0,C 180,E1 -6250.699,E2 -6250.699} C_VEL
LIN {X 0,Y 495.731,Z 364.737,A -85,B 0,C 180,E1 -6253.695,E2 -6253.695} C_VEL
LIN {X 0,Y 495.73,Z 364.73,A -85,B 0,C 180,E1 -6256.304,E2 -6256.304} C_VEL
LIN {X 0,Y 495.775,Z 364.73,A -85,B 0,C 180,E1 -6259.301,E2 -6259.301} C_VEL
LIN {X 0,Y 495.726,Z 364.73,A -85,B 0,C 180,E1 -6262.438,E2 -6262.438} C_VEL
LIN {X 0,Y 495.78,Z 364.732,A -85,B 0,C 180,E1 -6265.457,E2 -6265.457} C_VEL
LIN {X 0,Y 495.753,Z 364.727,A -85,B 0,C 180,E1 -6268.363,E2 -6268.363} C_VEL
LIN {X 0,Y 495.783,Z 364.729,A -85,B 0,C 180,E1 -6271.506,E2 -6271.506} C_VEL
LIN {X 0,Y 495.792,Z 364.723,A -85,B 0,C 180,E1 -6273.932,E2 -6273.932} C_VEL
LIN {X 0,Y 495.757,Z 364.734,A -85,B 0,C 180,E1 -6277.137,E2 -6277.137} C_VEL
LIN {X 0,Y 495.77,Z 364.725,A -85,B 0,C 180,E1 -6280.11,E2 -6280.11} C_VEL
LIN {X 0,Y 495.78,Z 364.726,A -85,B 0,C 180,E1 -6282.681,E2 -6282.681} C_VEL
LIN {X 0,Y 495.781,Z 364.731,A -85,B 0,C 180,E1 -6285.217,E2 -6285.217} C_VEL
LIN {X 0,Y 495.868,Z 364.714,A -85,B 0,C 180,E1 -6288.555,E2 -6288.555} C_VEL
LIN {X 0,Y 495.865,Z 364.713,A -85,B 0,C 180,E1 -6291.852,E2 -6291.852} C_VEL
LIN {X 0,Y 495.889,Z 364.711,A -85,B 0,C 180,E1 -6294.306,E2 -6294.306} C_VEL
LIN {X 0,Y 495.986,Z 364.699,A -85,B 0,C 180,E1 -6297.564,E2 -6297.564} C_VEL
LIN {X 0,Y 495.988,Z 364.698,A -85,B 0,C 180,E1 -6300,E2 -6300} C_VEL
LIN {X 0,Y 495.986,Z 364.7,A -85,B 0,C 180,E1 -6302.436,E2 -6302.436} C_VEL
LIN {X 0,Y 495.896,Z 364.709,A -85,B 0,C 180,E1 -6305.694,E2 -6305.694} C_VEL
LIN {X 0,Y 495.865,Z 364.714,A -85,B 0,C 180,E1 -6308.148,E2 -6308.148} C_VEL
LIN {X 0,Y 495.86,Z 364.714,A -85,B 0,C 180,E1 -6311.445,E2 -6311.445} C_VEL
LIN {X 0,Y 495.786,Z 364.731,A -85,B 0,C 180,E1 -6314.783,E2 -6314.783} C_VEL
LIN {X 0,Y 495.78,Z 364.725,A -85,B 0,C 180,E1 -6317.319,E2 -6317.319} C_VEL
LIN {X 0,Y 495.77,Z 364.725,A -85,B 0,C 180,E1 -6319.891,E2 -6319.891} C_VEL
LIN {X 0,Y 495.757,Z 364.732,A -85,B 0,C 180,E1 -6322.863,E2 -6322.863} C_VEL
LIN {X 0,Y 495.792,Z 364.724,A -85,B 0,C 180,E1 -6326.068,E2 -6326.068} C_VEL
LIN {X 0,Y 495.765,Z 364.73,A -85,B 0,C 180,E1 -6328.815,E2 -6328.815} C_VEL
LIN {X 0,Y 495.752,Z 364.727,A -85,B 0,C 180,E1 -6331.727,E2 -6331.727} C_VEL
LIN {X 0,Y 495.768,Z 364.73,A -85,B 0,C 180,E1 -6334.696,E2 -6334.696} C_VEL
LIN {X 0,Y 495.726,Z 364.73,A -85,B 0,C 180,E1 -6337.562,E2 -6337.562} C_VEL
LIN {X 0,Y 495.775,Z 364.728,A -85,B 0,C 180,E1 -6340.699,E2 -6340.699} C_VEL
LIN {X 0,Y 495.731,Z 364.731,A -85,B 0,C 180,E1 -6343.696,E2 -6343.696} C_VEL
LIN {X 0,Y 495.725,Z 364.739,A -85,B 0,C 180,E1 -6346.306,E2 -6346.306} C_VEL
LIN {X 0,Y 495.764,Z 364.725,A -85,B 0,C 180,E1 -6349.301,E2 -6349.301} C_VEL
LIN {X 0,Y 495.73,Z 364.735,A -85,B 0,C 180,E1 -6352.439,E2 -6352.439} C_VEL
LIN {X 0,Y 495.784,Z 364.724,A -85,B 0,C 180,E1 -6355.458,E2 -6355.458} C_VEL
LIN {X 0,Y 495.756,Z 364.732,A -85,B 0,C 180,E1 -6358.365,E2 -6358.365} C_VEL
LIN {X 0,Y 495.755,Z 364.728,A -85,B 0,C 180,E1 -6360.776,E2 -6360.776} C_VEL
LIN {X 0,Y 495.098,Z 364.81,A -85,B 0,C 180,E1 -6361.455,E2 -6361.455} C_VEL
LIN {X 0,Y 492.24,Z 365.167,A -85,B 0,C 180,E1 -6362.558,E2 -6362.558} C_VEL
LIN {X 0,Y 489.825,Z 365.467,A -85,B 0,C 180,E1 -6363.446,E2 -6363.446} C_VEL
LIN {X 0,Y 488.801,Z 365.601,A -85,B 0,C 180,E1 -6364.133,E2 -6364.133} C_VEL
LIN {X 0,Y 488.725,Z 365.608,A -85,B 0,C 180,E1 -6364.365,E2 -6364.365} C_VEL
LIN {X 0,Y 488.723,Z 365.606,A -85,B 0,C 180,E1 -6367.154,E2 -6367.154} C_VEL
LIN {X 0,Y 488.779,Z 365.801,A -85,B 0,C 180,E1 -6369.328,E2 -6369.328} C_VEL
LIN {X 0,Y 489.824,Z 372.018,A -85,B 0,C 180,E1 -6370.731,E2 -6370.731} C_VEL
LIN {X 0,Y 489.334,Z 386.429,A -85,B 0,C 180,E1 -6373.771,E2 -6373.771} C_VEL
LIN {X 0,Y 491.845,Z 399.196,A -85,B 0,C 180,E1 -6374.072,E2 -6374.072} C_VEL
LIN {X 0,Y 491.215,Z 493.463,A -85,B 0,C 180,E1 -6375.474,E2 -6375.474} C_VEL
LIN {X 0,Y 490.922,Z 506.591,A -85,B 0,C 180,E1 -6375.835,E2 -6375.835} C_VEL
LIN {X 0,Y 490.663,Z 518.655,A -85,B 0,C 180,E1 -6376.33,E2 -6376.33} C_VEL
LIN {X 0,Y 490.375,Z 529.372,A -85,B 0,C 180,E1 -6376.915,E2 -6376.915} C_VEL
LIN {X 0,Y 489.99,Z 540.406,A -85,B 0,C 180,E1 -6377.681,E2 -6377.681} C_VEL
LIN {X 0,Y 489.525,Z 551.087,A -85,B 0,C 180,E1 -6378.615,E2 -6378.615} C_VEL
LIN {X 0,Y 489.163,Z 560.693,A -85,B 0,C 180,E1 -6379.654,E2 -6379.654} C_VEL
LIN {X 0,Y 488.835,Z 568.56,A -85,B 0,C 180,E1 -6380.692,E2 -6380.692} C_VEL
LIN {X 0,Y 488.512,Z 576.251,A -85,B 0,C 180,E1 -6381.937,E2 -6381.937} C_VEL
LIN {X 0,Y 488.251,Z 583.304,A -85,B 0,C 180,E1 -6383.388,E2 -6383.388} C_VEL
LIN {X 0,Y 488.075,Z 588.004,A -85,B 0,C 180,E1 -6384.63,E2 -6384.63} C_VEL
LIN {X 0,Y 488.089,Z 591.597,A -85,B 0,C 180,E1 -6385.872,E2 -6385.872} C_VEL
LIN {X 0,Y 487.98,Z 593.46,A -85,B 0,C 180,E1 -6386.698,E2 -6386.698} C_VEL
LIN {X 0,Y 487.96,Z 594.862,A -85,B 0,C 180,E1 -6387.524,E2 -6387.524} C_VEL
LIN {X 0,Y 487.834,Z 596.476,A -85,B 0,C 180,E1 -6389.175,E2 -6389.175} C_VEL
LIN {X 0,Y 487.821,Z 596.712,A -85,B 0,C 180,E1 -6390,E2 -6390} C_VEL
LIN {X 0,Y 487.834,Z 596.527,A -85,B 0,C 180,E1 -6390.825,E2 -6390.825} C_VEL
LIN {X 0,Y 487.96,Z 594.98,A -85,B 0,C 180,E1 -6392.476,E2 -6392.476} C_VEL
LIN {X 0,Y 487.98,Z 593.629,A -85,B 0,C 180,E1 -6393.302,E2 -6393.302} C_VEL
LIN {X 0,Y 488.053,Z 590.772,A -85,B 0,C 180,E1 -6394.543,E2 -6394.543} C_VEL
LIN {X 0,Y 488.191,Z 586.897,A -85,B 0,C 180,E1 -6395.783,E2 -6395.783} C_VEL
LIN {X 0,Y 488.323,Z 581.899,A -85,B 0,C 180,E1 -6397.026,E2 -6397.026} C_VEL
LIN {X 0,Y 488.503,Z 575.606,A -85,B 0,C 180,E1 -6398.272,E2 -6398.272} C_VEL
LIN {X 0,Y 488.823,Z 567.723,A -85,B 0,C 180,E1 -6399.517,E2 -6399.517} C_VEL
LIN {X 0,Y 489.131,Z 559.687,A -85,B 0,C 180,E1 -6400.556,E2 -6400.556} C_VEL
LIN {X 0,Y 489.593,Z 549.874,A -85,B 0,C 180,E1 -6401.593,E2 -6401.593} C_VEL
LIN {X 0,Y 490.047,Z 539.053,A -85,B 0,C 180,E1 -6402.512,E2 -6402.512} C_VEL
LIN {X 0,Y 490.4,Z 528.027,A -85,B 0,C 180,E1 -6403.255,E2 -6403.255} C_VEL
LIN {X 0,Y 490.729,Z 516.082,A -85,B 0,C 180,E1 -6403.879,E2 -6403.879} C_VEL
LIN {X 0,Y 491.05,Z 502.994,A -85,B 0,C 180,E1 -6404.372,E2 -6404.372} C_VEL
LIN {X 0,Y 491.246,Z 489.849,A -85,B 0,C 180,E1 -6404.684,E2 -6404.684} C_VEL
LIN {X 0,Y 491.75,Z 398.668,A -85,B 0,C 180,E1 -6406.03,E2 -6406.03} C_VEL
LIN {X 0,Y 489.329,Z 386.499,A -85,B 0,C 180,E1 -6406.307,E2 -6406.307} C_VEL
LIN {X 0,Y 489.865,Z 372.447,A -85,B 0,C 180,E1 -6409.267,E2 -6409.267} C_VEL
LIN {X 0,Y 488.716,Z 365.611,A -85,B 0,C 180,E1 -6410.814,E2 -6410.814} C_VEL
LIN {X 0,Y 488.696,Z 365.617,A -85,B 0,C 180,E1 -6413.745,E2 -6413.745} C_VEL
LIN {X 0,Y 488.793,Z 365.594,A -85,B 0,C 180,E1 -6416.943,E2 -6416.943} C_VEL
LIN {X 0,Y 488.71,Z 365.607,A -85,B 0,C 180,E1 -6420.362,E2 -6420.362} C_VEL
LIN {X 0,Y 488.735,Z 365.604,A -85,B 0,C 180,E1 -6423.484,E2 -6423.484} C_VEL
LIN {X 0,Y 488.688,Z 365.609,A -85,B 0,C 180,E1 -6426.355,E2 -6426.355} C_VEL
LIN {X 0,Y 488.699,Z 365.607,A -85,B 0,C 180,E1 -6429.253,E2 -6429.253} C_VEL
LIN {X 0,Y 488.704,Z 365.611,A -85,B 0,C 180,E1 -6431.599,E2 -6431.599} C_VEL
LIN {X 0,Y 488.708,Z 365.604,A -85,B 0,C 180,E1 -6434.801,E2 -6434.801} C_VEL
LIN {X 0,Y 488.727,Z 365.607,A -85,B 0,C 180,E1 -6437.478,E2 -6437.478} C_VEL
LIN {X 0,Y 488.737,Z 365.601,A -85,B 0,C 180,E1 -6440.749,E2 -6440.749} C_VEL
LIN {X 0,Y 488.681,Z 365.613,A -85,B 0,C 180,E1 -6443.868,E2 -6443.868} C_VEL
LIN {X 0,Y 488.733,Z 365.602,A -85,B 0,C 180,E1 -6446.877,E2 -6446.877} C_VEL
LIN {X 0,Y 488.717,Z 365.608,A -85,B 0,C 180,E1 -6449.78,E2 -6449.78} C_VEL
LIN {X 0,Y 488.792,Z 365.597,A -85,B 0,C 180,E1 -6453.054,E2 -6453.054} C_VEL
LIN {X 0,Y 488.693,Z 365.607,A -85,B 0,C 180,E1 -6456.254,E2 -6456.254} C_VEL
LIN {X 0,Y 488.739,Z 365.606,A -85,B 0,C 180,E1 -6459.175,E2 -6459.175} C_VEL
LIN {X 0,Y 488.727,Z 365.602,A -85,B 0,C 180,E1 -6462.423,E2 -6462.423} C_VEL
LIN {X 0,Y 488.756,Z 365.603,A -85,B 0,C 180,E1 -6464.999,E2 -6464.999} C_VEL
LIN {X 0,Y 488.822,Z 365.59,A -85,B 0,C 180,E1 -6468.388,E2 -6468.388} C_VEL
LIN {X 0,Y 488.81,Z 365.594,A -85,B 0,C 180,E1 -6471.733,E2 -6471.733} C_VEL
LIN {X 0,Y 488.847,Z 365.587,A -85,B 0,C 180,E1 -6474.224,E2 -6474.224} C_VEL
LIN {X 0,Y 488.954,Z 365.577,A -85,B 0,C 180,E1 -6477.529,E2 -6477.529} C_VEL
LIN {X 0,Y 488.96,Z 365.573,A -85,B 0,C 180,E1 -6480,E2 -6480} C_VEL
LIN {X 0,Y 488.954,Z 365.575,A -85,B 0,C 180,E1 -6482.471,E2 -6482.471} C_VEL
LIN {X 0,Y 488.854,Z 365.587,A -85,B 0,C 180,E1 -6485.776,E2 -6485.776} C_VEL
LIN {X 0,Y 488.81,Z 365.592,A -85,B 0,C 180,E1 -6488.267,E2 -6488.267} C_VEL
LIN {X 0,Y 488.825,Z 365.591,A -85,B 0,C 180,E1 -6491.612,E2 -6491.612} C_VEL
LIN {X 0,Y 488.753,Z 365.606,A -85,B 0,C 180,E1 -6495.001,E2 -6495.001} C_VEL
LIN {X 0,Y 488.746,Z 365.603,A -85,B 0,C 180,E1 -6498.443,E2 -6498.443} C_VEL
LIN {X 0,Y 488.704,Z 365.61,A -85,B 0,C 180,E1 -6501.071,E2 -6501.071} C_VEL
LIN {X 0,Y 488.693,Z 365.606,A -85,B 0,C 180,E1 -6503.746,E2 -6503.746} C_VEL
LIN {X 0,Y 488.791,Z 365.599,A -85,B 0,C 180,E1 -6506.946,E2 -6506.946} C_VEL
LIN {X 0,Y 488.703,Z 365.609,A -85,B 0,C 180,E1 -6510.364,E2 -6510.364} C_VEL
LIN {X 0,Y 488.73,Z 365.602,A -85,B 0,C 180,E1 -6513.485,E2 -6513.485} C_VEL
LIN {X 0,Y 488.683,Z 365.613,A -85,B 0,C 180,E1 -6516.356,E2 -6516.356} C_VEL
LIN {X 0,Y 488.737,Z 365.602,A -85,B 0,C 180,E1 -6519.251,E2 -6519.251} C_VEL
LIN {X 0,Y 488.731,Z 365.61,A -85,B 0,C 180,E1 -6522.522,E2 -6522.522} C_VEL
LIN {X 0,Y 488.698,Z 365.608,A -85,B 0,C 180,E1 -6525.977,E2 -6525.977} C_VEL
LIN {X 0,Y 488.716,Z 365.61,A -85,B 0,C 180,E1 -6528.586,E2 -6528.586} C_VEL
LIN {X 0,Y 488.679,Z 365.61,A -85,B 0,C 180,E1 -6531.801,E2 -6531.801} C_VEL
LIN {X 0,Y 488.727,Z 365.603,A -85,B 0,C 180,E1 -6535.052,E2 -6535.052} C_VEL
LIN {X 0,Y 488.705,Z 365.61,A -85,B 0,C 180,E1 -6538.046,E2 -6538.046} C_VEL
LIN {X 0,Y 488.723,Z 365.607,A -85,B 0,C 180,E1 -6540.73,E2 -6540.73} C_VEL
LIN {X 0,Y 488.759,Z 365.605,A -85,B 0,C 180,E1 -6543.529,E2 -6543.529} C_VEL
LIN {X 0,Y 488.814,Z 365.777,A -85,B 0,C 180,E1 -6544.449,E2 -6544.449} C_VEL
LIN {X 0,Y 490.761,Z 376.663,A -85,B 0,C 180,E1 -6546.423,E2 -6546.423} C_VEL
LIN {X 0,Y 490.241,Z 392.001,A -85,B 0,C 180,E1 -6548.999,E2 -6548.999} C_VEL
LIN {X 0,Y 489.565,Z 411.559,A -85,B 0,C 180,E1 -6552.239,E2 -6552.239} C_VEL
LIN {X 0,Y 489.3,Z 420.558,A -85,B 0,C 180,E1 -6553.725,E2 -6553.725} C_VEL
LIN {X 0,Y 491.712,Z 436.674,A -85,B 0,C 180,E1 -6554.05,E2 -6554.05} C_VEL
LIN {X 0,Y 491.118,Z 528.905,A -85,B 0,C 180,E1 -6555.418,E2 -6555.418} C_VEL
LIN {X 0,Y 490.788,Z 542.188,A -85,B 0,C 180,E1 -6555.779,E2 -6555.779} C_VEL
LIN {X 0,Y 490.423,Z 554.362,A -85,B 0,C 180,E1 -6556.27,E2 -6556.27} C_VEL
LIN {X 0,Y 490.039,Z 566.654,A -85,B 0,C 180,E1 -6556.946,E2 -6556.946} C_VEL
LIN {X 0,Y 489.554,Z 578.263,A -85,B 0,C 180,E1 -6557.775,E2 -6557.775} C_VEL
LIN {X 0,Y 489.223,Z 588.725,A -85,B 0,C 180,E1 -6558.713,E2 -6558.713} C_VEL
LIN {X 0,Y 488.849,Z 597.277,A -85,B 0,C 180,E1 -6559.647,E2 -6559.647} C_VEL
LIN {X 0,Y 488.548,Z 605.171,A -85,B 0,C 180,E1 -6560.687,E2 -6560.687} C_VEL
LIN {X 0,Y 488.28,Z 612.882,A -85,B 0,C 180,E1 -6561.933,E2 -6561.933} C_VEL
LIN {X 0,Y 488.1,Z 619.994,A -85,B 0,C 180,E1 -6563.386,E2 -6563.386} C_VEL
LIN {X 0,Y 488.019,Z 624.727,A -85,B 0,C 180,E1 -6564.629,E2 -6564.629} C_VEL
LIN {X 0,Y 487.929,Z 628.341,A -85,B 0,C 180,E1 -6565.87,E2 -6565.87} C_VEL
LIN {X 0,Y 487.964,Z 630.209,A -85,B 0,C 180,E1 -6566.697,E2 -6566.697} C_VEL
LIN {X 0,Y 487.891,Z 632.604,A -85,B 0,C 180,E1 -6568.349,E2 -6568.349} C_VEL
LIN {X 0,Y 487.819,Z 633.428,A -85,B 0,C 180,E1 -6570,E2 -6570} C_VEL
LIN {X 0,Y 487.891,Z 632.606,A -85,B 0,C 180,E1 -6571.651,E2 -6571.651} C_VEL
LIN {X 0,Y 487.964,Z 630.212,A -85,B 0,C 180,E1 -6573.303,E2 -6573.303} C_VEL
LIN {X 0,Y 487.921,Z 627.269,A -85,B 0,C 180,E1 -6574.544,E2 -6574.544} C_VEL
LIN {X 0,Y 488.025,Z 623.289,A -85,B 0,C 180,E1 -6575.785,E2 -6575.785} C_VEL
LIN {X 0,Y 488.182,Z 617.169,A -85,B 0,C 180,E1 -6577.236,E2 -6577.236} C_VEL
LIN {X 0,Y 488.363,Z 610.48,A -85,B 0,C 180,E1 -6578.482,E2 -6578.482} C_VEL
LIN {X 0,Y 488.656,Z 602.184,A -85,B 0,C 180,E1 -6579.729,E2 -6579.729} C_VEL
LIN {X 0,Y 489.005,Z 593.685,A -85,B 0,C 180,E1 -6580.768,E2 -6580.768} C_VEL
LIN {X 0,Y 489.449,Z 583.186,A -85,B 0,C 180,E1 -6581.807,E2 -6581.807} C_VEL
LIN {X 0,Y 489.76,Z 572.912,A -85,B 0,C 180,E1 -6582.632,E2 -6582.632} C_VEL
LIN {X 0,Y 490.229,Z 561.417,A -85,B 0,C 180,E1 -6583.366,E2 -6583.366} C_VEL
LIN {X 0,Y 490.575,Z 549.747,A -85,B 0,C 180,E1 -6583.937,E2 -6583.937} C_VEL
LIN {X 0,Y 490.947,Z 536.305,A -85,B 0,C 180,E1 -6584.402,E2 -6584.402} C_VEL
LIN {X 0,Y 491.218,Z 523.039,A -85,B 0,C 180,E1 -6584.685,E2 -6584.685} C_VEL
LIN {X 0,Y 491.61,Z 435.469,A -85,B 0,C 180,E1 -6585.971,E2 -6585.971} C_VEL
LIN {X 0,Y 489.29,Z 420.558,A -85,B 0,C 180,E1 -6586.277,E2 -6586.277} C_VEL
LIN {X 0,Y 489.863,Z 402.438,A -85,B 0,C 180,E1 -6589.267,E2 -6589.267} C_VEL
LIN {X 0,Y 490.638,Z 382.843,A -85,B 0,C 180,E1 -6592.53,E2 -6592.53} C_VEL
LIN {X 0,Y 490.748,Z 376.295,A -85,B 0,C 180,E1 -6593.639,E2 -6593.639} C_VEL
LIN {X 0,Y 488.789,Z 365.603,A -85,B 0,C 180,E1 -6595.61,E2 -6595.61} C_VEL
LIN {X 0,Y 488.745,Z 365.605,A -85,B 0,C 180,E1 -6598.328,E2 -6598.328} C_VEL
LIN {X 0,Y 488.694,Z 365.611,A -85,B 0,C 180,E1 -6601.179,E2 -6601.179} C_VEL
LIN {X 0,Y 488.734,Z 365.604,A -85,B 0,C 180,E1 -6604.112,E2 -6604.112} C_VEL
LIN {X 0,Y 488.681,Z 365.61,A -85,B 0,C 180,E1 -6607.158,E2 -6607.158} C_VEL
LIN {X 0,Y 488.715,Z 365.604,A -85,B 0,C 180,E1 -6610.344,E2 -6610.344} C_VEL
LIN {X 0,Y 488.712,Z 365.604,A -85,B 0,C 180,E1 -6612.826,E2 -6612.826} C_VEL
LIN {X 0,Y 488.698,Z 365.609,A -85,B 0,C 180,E1 -6615.975,E2 -6615.975} C_VEL
LIN {X 0,Y 488.72,Z 365.603,A -85,B 0,C 180,E1 -6618.585,E2 -6618.585} C_VEL
LIN {X 0,Y 488.735,Z 365.603,A -85,B 0,C 180,E1 -6620.941,E2 -6620.941} C_VEL
LIN {X 0,Y 488.679,Z 365.611,A -85,B 0,C 180,E1 -6623.868,E2 -6623.868} C_VEL
LIN {X 0,Y 488.733,Z 365.603,A -85,B 0,C 180,E1 -6626.877,E2 -6626.877} C_VEL
LIN {X 0,Y 488.727,Z 365.605,A -85,B 0,C 180,E1 -6629.781,E2 -6629.781} C_VEL
LIN {X 0,Y 488.791,Z 365.599,A -85,B 0,C 180,E1 -6633.054,E2 -6633.054} C_VEL
LIN {X 0,Y 488.693,Z 365.606,A -85,B 0,C 180,E1 -6636.254,E2 -6636.254} C_VEL
LIN {X 0,Y 488.739,Z 365.609,A -85,B 0,C 180,E1 -6639.175,E2 -6639.175} C_VEL
LIN {X 0,Y 488.75,Z 365.602,A -85,B 0,C 180,E1 -6641.627,E2 -6641.627} C_VEL
LIN {X 0,Y 488.753,Z 365.605,A -85,B 0,C 180,E1 -6644.999,E2 -6644.999} C_VEL
LIN {X 0,Y 488.825,Z 365.591,A -85,B 0,C 180,E1 -6648.388,E2 -6648.388} C_VEL
LIN {X 0,Y 488.81,Z 365.593,A -85,B 0,C 180,E1 -6651.733,E2 -6651.733} C_VEL
LIN {X 0,Y 488.848,Z 365.587,A -85,B 0,C 180,E1 -6654.224,E2 -6654.224} C_VEL
LIN {X 0,Y 488.954,Z 365.576,A -85,B 0,C 180,E1 -6657.529,E2 -6657.529} C_VEL
LIN {X 0,Y 488.96,Z 365.573,A -85,B 0,C 180,E1 -6660,E2 -6660} C_VEL
LIN {X 0,Y 488.954,Z 365.577,A -85,B 0,C 180,E1 -6662.471,E2 -6662.471} C_VEL
LIN {X 0,Y 488.854,Z 365.586,A -85,B 0,C 180,E1 -6665.776,E2 -6665.776} C_VEL
LIN {X 0,Y 488.81,Z 365.594,A -85,B 0,C 180,E1 -6668.267,E2 -6668.267} C_VEL
LIN {X 0,Y 488.822,Z 365.591,A -85,B 0,C 180,E1 -6671.612,E2 -6671.612} C_VEL
LIN {X 0,Y 488.756,Z 365.603,A -85,B 0,C 180,E1 -6675.001,E2 -6675.001} C_VEL
LIN {X 0,Y 488.746,Z 365.605,A -85,B 0,C 180,E1 -6678.443,E2 -6678.443} C_VEL
LIN {X 0,Y 488.704,Z 365.608,A -85,B 0,C 180,E1 -6681.071,E2 -6681.071} C_VEL
LIN {X 0,Y 488.693,Z 365.606,A -85,B 0,C 180,E1 -6683.746,E2 -6683.746} C_VEL
LIN {X 0,Y 488.792,Z 365.598,A -85,B 0,C 180,E1 -6686.946,E2 -6686.946} C_VEL
LIN {X 0,Y 488.703,Z 365.611,A -85,B 0,C 180,E1 -6690.364,E2 -6690.364} C_VEL
LIN {X 0,Y 488.729,Z 365.602,A -85,B 0,C 180,E1 -6693.485,E2 -6693.485} C_VEL
LIN {X 0,Y 488.682,Z 365.615,A -85,B 0,C 180,E1 -6696.356,E2 -6696.356} C_VEL
LIN {X 0,Y 488.737,Z 365.601,A -85,B 0,C 180,E1 -6699.251,E2 -6699.251} C_VEL
LIN {X 0,Y 488.727,Z 365.608,A -85,B 0,C 180,E1 -6702.522,E2 -6702.522} C_VEL
LIN {X 0,Y 488.708,Z 365.605,A -85,B 0,C 180,E1 -6705.199,E2 -6705.199} C_VEL
LIN {X 0,Y 488.704,Z 365.612,A -85,B 0,C 180,E1 -6708.401,E2 -6708.401} C_VEL
LIN {X 0,Y 488.702,Z 365.606,A -85,B 0,C 180,E1 -6710.948,E2 -6710.948} C_VEL
LIN {X 0,Y 488.684,Z 365.611,A -85,B 0,C 180,E1 -6713.87,E2 -6713.87} C_VEL
LIN {X 0,Y 488.738,Z 365.601,A -85,B 0,C 180,E1 -6716.878,E2 -6716.878} C_VEL
LIN {X 0,Y 488.725,Z 365.606,A -85,B 0,C 180,E1 -6719.782,E2 -6719.782} C_VEL
LIN {X 0,Y 488.793,Z 365.594,A -85,B 0,C 180,E1 -6723.057,E2 -6723.057} C_VEL
LIN {X 0,Y 488.725,Z 365.608,A -85,B 0,C 180,E1 -6724.365,E2 -6724.365} C_VEL
LIN {X 0,Y 488.075,Z 365.695,A -85,B 0,C 180,E1 -6725.053,E2 -6725.053} C_VEL
LIN {X 0,Y 485.212,Z 366.053,A -85,B 0,C 180,E1 -6726.17,E2 -6726.17} C_VEL
LIN {X 0,Y 482.775,Z 366.353,A -85,B 0,C 180,E1 -6727.07,E2 -6727.07} C_VEL
LIN {X 0,Y 481.724,Z 366.482,A -85,B 0,C 180,E1 -6727.765,E2 -6727.765} C_VEL
LIN {X 0,Y 481.636,Z 366.491,A -85,B 0,C 180,E1 -6728.001,E2 -6728.001} C_VEL
LIN {X 0,Y 481.728,Z 366.562,A -85,B 0,C 180,E1 -6729.134,E2 -6729.134} C_VEL
LIN {X 0,Y 482.729,Z 372.248,A -85,B 0,C 180,E1 -6730.437,E2 -6730.437} C_VEL
LIN {X 0,Y 482.698,Z 378.335,A -85,B 0,C 180,E1 -6731.758,E2 -6731.758} C_VEL
LIN {X 0,Y 482.385,Z 386.745,A -85,B 0,C 180,E1 -6733.544,E2 -6733.544} C_VEL
LIN {X 0,Y 485.01,Z 400.48,A -85,B 0,C 180,E1 -6733.856,E2 -6733.856} C_VEL
LIN {X 0,Y 484.372,Z 493.751,A -85,B 0,C 180,E1 -6735.264,E2 -6735.264} C_VEL
LIN {X 0,Y 484.06,Z 507.631,A -85,B 0,C 180,E1 -6735.657,E2 -6735.657} C_VEL
LIN {X 0,Y 483.775,Z 520.04,A -85,B 0,C 180,E1 -6736.185,E2 -6736.185} C_VEL
LIN {X 0,Y 483.395,Z 531.65,A -85,B 0,C 180,E1 -6736.853,E2 -6736.853} C_VEL
LIN {X 0,Y 482.986,Z 543.249,A -85,B 0,C 180,E1 -6737.713,E2 -6737.713} C_VEL
LIN {X 0,Y 482.495,Z 553.483,A -85,B 0,C 180,E1 -6738.66,E2 -6738.66} C_VEL
LIN {X 0,Y 482.097,Z 562.661,A -85,B 0,C 180,E1 -6739.713,E2 -6739.713} C_VEL
LIN {X 0,Y 481.688,Z 571.568,A -85,B 0,C 180,E1 -6740.976,E2 -6740.976} C_VEL
LIN {X 0,Y 481.372,Z 578.738,A -85,B 0,C 180,E1 -6742.239,E2 -6742.239} C_VEL
LIN {X 0,Y 481.173,Z 584.824,A -85,B 0,C 180,E1 -6743.594,E2 -6743.594} C_VEL
LIN {X 0,Y 480.92,Z 589.588,A -85,B 0,C 180,E1 -6744.97,E2 -6744.97} C_VEL
LIN {X 0,Y 481.009,Z 591.866,A -85,B 0,C 180,E1 -6745.811,E2 -6745.811} C_VEL
LIN {X 0,Y 480.912,Z 593.727,A -85,B 0,C 180,E1 -6746.649,E2 -6746.649} C_VEL
LIN {X 0,Y 480.87,Z 595.129,A -85,B 0,C 180,E1 -6747.487,E2 -6747.487} C_VEL
LIN {X 0,Y 480.76,Z 596.743,A -85,B 0,C 180,E1 -6749.162,E2 -6749.162} C_VEL
LIN {X 0,Y 480.745,Z 596.979,A -85,B 0,C 180,E1 -6750,E2 -6750} C_VEL
LIN {X 0,Y 480.76,Z 596.793,A -85,B 0,C 180,E1 -6750.838,E2 -6750.838} C_VEL
LIN {X 0,Y 480.87,Z 595.246,A -85,B 0,C 180,E1 -6752.513,E2 -6752.513} C_VEL
LIN {X 0,Y 480.912,Z 593.894,A -85,B 0,C 180,E1 -6753.351,E2 -6753.351} C_VEL
LIN {X 0,Y 480.972,Z 591.038,A -85,B 0,C 180,E1 -6754.61,E2 -6754.61} C_VEL
LIN {X 0,Y 481.141,Z 587.161,A -85,B 0,C 180,E1 -6755.869,E2 -6755.869} C_VEL
LIN {X 0,Y 481.276,Z 582.162,A -85,B 0,C 180,E1 -6757.13,E2 -6757.13} C_VEL
LIN {X 0,Y 481.489,Z 575.869,A -85,B 0,C 180,E1 -6758.393,E2 -6758.393} C_VEL
LIN {X 0,Y 481.834,Z 567.986,A -85,B 0,C 180,E1 -6759.656,E2 -6759.656} C_VEL
LIN {X 0,Y 482.206,Z 558.179,A -85,B 0,C 180,E1 -6760.922,E2 -6760.922} C_VEL
LIN {X 0,Y 482.78,Z 547.881,A -85,B 0,C 180,E1 -6761.972,E2 -6761.972} C_VEL
LIN {X 0,Y 483.165,Z 536.931,A -85,B 0,C 180,E1 -6762.873,E2 -6762.873} C_VEL
LIN {X 0,Y 483.569,Z 526.525,A -85,B 0,C 180,E1 -6763.553,E2 -6763.553} C_VEL
LIN {X 0,Y 483.931,Z 513.981,A -85,B 0,C 180,E1 -6764.186,E2 -6764.186} C_VEL
LIN {X 0,Y 484.253,Z 500.5,A -85,B 0,C 180,E1 -6764.659,E2 -6764.659} C_VEL
LIN {X 0,Y 484.401,Z 486.999,A -85,B 0,C 180,E1 -6764.95,E2 -6764.95} C_VEL
LIN {X 0,Y 484.957,Z 399.599,A -85,B 0,C 180,E1 -6766.25,E2 -6766.25} C_VEL
LIN {X 0,Y 482.394,Z 386.75,A -85,B 0,C 180,E1 -6766.548,E2 -6766.548} C_VEL
LIN {X 0,Y 482.886,Z 374.548,A -85,B 0,C 180,E1 -6769.145,E2 -6769.145} C_VEL
LIN {X 0,Y 482.496,Z 370.652,A -85,B 0,C 180,E1 -6770.016,E2 -6770.016} C_VEL
LIN {X 0,Y 481.667,Z 366.489,A -85,B 0,C 180,E1 -6771.007,E2 -6771.007} C_VEL
LIN {X 0,Y 481.679,Z 366.489,A -85,B 0,C 180,E1 -6774.112,E2 -6774.112} C_VEL
LIN {X 0,Y 481.748,Z 366.472,A -85,B 0,C 180,E1 -6777.139,E2 -6777.139} C_VEL
LIN {X 0,Y 481.679,Z 366.485,A -85,B 0,C 180,E1 -6779.74,E2 -6779.74} C_VEL
LIN {X 0,Y 481.672,Z 366.482,A -85,B 0,C 180,E1 -6782.673,E2 -6782.673} C_VEL
LIN {X 0,Y 481.642,Z 366.491,A -85,B 0,C 180,E1 -6785.708,E2 -6785.708} C_VEL
LIN {X 0,Y 481.669,Z 366.481,A -85,B 0,C 180,E1 -6788.858,E2 -6788.858} C_VEL
LIN {X 0,Y 481.649,Z 366.491,A -85,B 0,C 180,E1 -6791.912,E2 -6791.912} C_VEL
LIN {X 0,Y 481.656,Z 366.484,A -85,B 0,C 180,E1 -6794.456,E2 -6794.456} C_VEL
LIN {X 0,Y 481.684,Z 366.48,A -85,B 0,C 180,E1 -6796.845,E2 -6796.845} C_VEL
LIN {X 0,Y 481.684,Z 366.483,A -85,B 0,C 180,E1 -6800.06,E2 -6800.06} C_VEL
LIN {X 0,Y 481.624,Z 366.49,A -85,B 0,C 180,E1 -6803.253,E2 -6803.253} C_VEL
LIN {X 0,Y 481.703,Z 366.478,A -85,B 0,C 180,E1 -6806.329,E2 -6806.329} C_VEL
LIN {X 0,Y 481.645,Z 366.491,A -85,B 0,C 180,E1 -6809.416,E2 -6809.416} C_VEL
LIN {X 0,Y 481.695,Z 366.479,A -85,B 0,C 180,E1 -6812.168,E2 -6812.168} C_VEL
LIN {X 0,Y 481.712,Z 366.478,A -85,B 0,C 180,E1 -6814.969,E2 -6814.969} C_VEL
LIN {X 0,Y 481.652,Z 366.488,A -85,B 0,C 180,E1 -6817.705,E2 -6817.705} C_VEL
LIN {X 0,Y 481.7,Z 366.477,A -85,B 0,C 180,E1 -6820.393,E2 -6820.393} C_VEL
LIN {X 0,Y 481.684,Z 366.484,A -85,B 0,C 180,E1 -6823.034,E2 -6823.034} C_VEL
LIN {X 0,Y 481.685,Z 366.483,A -85,B 0,C 180,E1 -6825.638,E2 -6825.638} C_VEL
LIN {X 0,Y 481.786,Z 366.467,A -85,B 0,C 180,E1 -6828.216,E2 -6828.216} C_VEL
LIN {X 0,Y 481.755,Z 366.474,A -85,B 0,C 180,E1 -6831.611,E2 -6831.611} C_VEL
LIN {X 0,Y 481.808,Z 366.464,A -85,B 0,C 180,E1 -6834.139,E2 -6834.139} C_VEL
LIN {X 0,Y 481.921,Z 366.454,A -85,B 0,C 180,E1 -6837.492,E2 -6837.492} C_VEL
LIN {X 0,Y 481.931,Z 366.449,A -85,B 0,C 180,E1 -6840,E2 -6840} C_VEL
LIN {X 0,Y 481.921,Z 366.452,A -85,B 0,C 180,E1 -6842.507,E2 -6842.507} C_VEL
LIN {X 0,Y 481.813,Z 366.464,A -85,B 0,C 180,E1 -6845.86,E2 -6845.86} C_VEL
LIN {X 0,Y 481.755,Z 366.472,A -85,B 0,C 180,E1 -6848.388,E2 -6848.388} C_VEL
LIN {X 0,Y 481.788,Z 366.467,A -85,B 0,C 180,E1 -6851.784,E2 -6851.784} C_VEL
LIN {X 0,Y 481.733,Z 366.477,A -85,B 0,C 180,E1 -6855.225,E2 -6855.225} C_VEL
LIN {X 0,Y 481.704,Z 366.484,A -85,B 0,C 180,E1 -6858.722,E2 -6858.722} C_VEL
LIN {X 0,Y 481.646,Z 366.486,A -85,B 0,C 180,E1 -6861.395,E2 -6861.395} C_VEL
LIN {X 0,Y 481.674,Z 366.482,A -85,B 0,C 180,E1 -6864.113,E2 -6864.113} C_VEL
LIN {X 0,Y 481.744,Z 366.475,A -85,B 0,C 180,E1 -6867.141,E2 -6867.141} C_VEL
LIN {X 0,Y 481.672,Z 366.481,A -85,B 0,C 180,E1 -6869.742,E2 -6869.742} C_VEL
LIN {X 0,Y 481.666,Z 366.49,A -85,B 0,C 180,E1 -6872.675,E2 -6872.675} C_VEL
LIN {X 0,Y 481.637,Z 366.485,A -85,B 0,C 180,E1 -6875.71,E2 -6875.71} C_VEL
LIN {X 0,Y 481.709,Z 366.477,A -85,B 0,C 180,E1 -6879.355,E2 -6879.355} C_VEL
LIN {X 0,Y 481.67,Z 366.485,A -85,B 0,C 180,E1 -6882.158,E2 -6882.158} C_VEL
LIN {X 0,Y 481.656,Z 366.492,A -85,B 0,C 180,E1 -6884.458,E2 -6884.458} C_VEL
LIN {X 0,Y 481.651,Z 366.485,A -85,B 0,C 180,E1 -6887.841,E2 -6887.841} C_VEL
LIN {X 0,Y 481.678,Z 366.485,A -85,B 0,C 180,E1 -6890.652,E2 -6890.652} C_VEL
LIN {X 0,Y 481.63,Z 366.486,A -85,B 0,C 180,E1 -6893.376,E2 -6893.376} C_VEL
LIN {X 0,Y 481.708,Z 366.485,A -85,B 0,C 180,E1 -6896.331,E2 -6896.331} C_VEL
LIN {X 0,Y 481.651,Z 366.484,A -85,B 0,C 180,E1 -6899.418,E2 -6899.418} C_VEL
LIN {X 0,Y 481.7,Z 366.485,A -85,B 0,C 180,E1 -6902.169,E2 -6902.169} C_VEL
LIN {X 0,Y 481.763,Z 366.554,A -85,B 0,C 180,E1 -6904.225,E2 -6904.225} C_VEL
LIN {X 0,Y 483.793,Z 377.419,A -85,B 0,C 180,E1 -6906.233,E2 -6906.233} C_VEL
LIN {X 0,Y 483.383,Z 390.76,A -85,B 0,C 180,E1 -6908.515,E2 -6908.515} C_VEL
LIN {X 0,Y 482.619,Z 411.307,A -85,B 0,C 180,E1 -6911.975,E2 -6911.975} C_VEL
LIN {X 0,Y 482.316,Z 420.524,A -85,B 0,C 180,E1 -6913.491,E2 -6913.491} C_VEL
LIN {X 0,Y 484.872,Z 437.567,A -85,B 0,C 180,E1 -6913.836,E2 -6913.836} C_VEL
LIN {X 0,Y 484.252,Z 528.644,A -85,B 0,C 180,E1 -6915.207,E2 -6915.207} C_VEL
LIN {X 0,Y 483.924,Z 541.925,A -85,B 0,C 180,E1 -6915.573,E2 -6915.573} C_VEL
LIN {X 0,Y 483.517,Z 554.098,A -85,B 0,C 180,E1 -6916.07,E2 -6916.07} C_VEL
LIN {X 0,Y 483.108,Z 566.388,A -85,B 0,C 180,E1 -6916.755,E2 -6916.755} C_VEL
LIN {X 0,Y 482.568,Z 578.072,A -85,B 0,C 180,E1 -6917.602,E2 -6917.602} C_VEL
LIN {X 0,Y 482.189,Z 588.456,A -85,B 0,C 180,E1 -6918.546,E2 -6918.546} C_VEL
LIN {X 0,Y 481.828,Z 597.009,A -85,B 0,C 180,E1 -6919.495,E2 -6919.495} C_VEL
LIN {X 0,Y 481.489,Z 604.902,A -85,B 0,C 180,E1 -6920.549,E2 -6920.549} C_VEL
LIN {X 0,Y 481.23,Z 612.614,A -85,B 0,C 180,E1 -6921.814,E2 -6921.814} C_VEL
LIN {X 0,Y 481.019,Z 619.726,A -85,B 0,C 180,E1 -6923.288,E2 -6923.288} C_VEL
LIN {X 0,Y 480.932,Z 624.459,A -85,B 0,C 180,E1 -6924.55,E2 -6924.55} C_VEL
LIN {X 0,Y 480.829,Z 628.073,A -85,B 0,C 180,E1 -6925.809,E2 -6925.809} C_VEL
LIN {X 0,Y 480.888,Z 629.942,A -85,B 0,C 180,E1 -6926.649,E2 -6926.649} C_VEL
LIN {X 0,Y 480.821,Z 632.338,A -85,B 0,C 180,E1 -6928.325,E2 -6928.325} C_VEL
LIN {X 0,Y 480.743,Z 633.162,A -85,B 0,C 180,E1 -6930,E2 -6930} C_VEL
LIN {X 0,Y 480.821,Z 632.34,A -85,B 0,C 180,E1 -6931.675,E2 -6931.675} C_VEL
LIN {X 0,Y 480.888,Z 629.946,A -85,B 0,C 180,E1 -6933.351,E2 -6933.351} C_VEL
LIN {X 0,Y 480.839,Z 627.001,A -85,B 0,C 180,E1 -6934.611,E2 -6934.611} C_VEL
LIN {X 0,Y 480.929,Z 623.021,A -85,B 0,C 180,E1 -6935.871,E2 -6935.871} C_VEL
LIN {X 0,Y 481.107,Z 616.9,A -85,B 0,C 180,E1 -6937.343,E2 -6937.343} C_VEL
LIN {X 0,Y 481.318,Z 610.212,A -85,B 0,C 180,E1 -6938.607,E2 -6938.607} C_VEL
LIN {X 0,Y 481.603,Z 601.915,A -85,B 0,C 180,E1 -6939.873,E2 -6939.873} C_VEL
LIN {X 0,Y 481.992,Z 593.416,A -85,B 0,C 180,E1 -6940.927,E2 -6940.927} C_VEL
LIN {X 0,Y 482.457,Z 582.937,A -85,B 0,C 180,E1 -6941.978,E2 -6941.978} C_VEL
LIN {X 0,Y 482.871,Z 571.599,A -85,B 0,C 180,E1 -6942.893,E2 -6942.893} C_VEL
LIN {X 0,Y 483.306,Z 561.147,A -85,B 0,C 180,E1 -6943.561,E2 -6943.561} C_VEL
LIN {X 0,Y 483.695,Z 549.477,A -85,B 0,C 180,E1 -6944.139,E2 -6944.139} C_VEL
LIN {X 0,Y 484.06,Z 536.949,A -85,B 0,C 180,E1 -6944.584,E2 -6944.584} C_VEL
LIN {X 0,Y 484.337,Z 524.279,A -85,B 0,C 180,E1 -6944.871,E2 -6944.871} C_VEL
LIN {X 0,Y 484.809,Z 436.605,A -85,B 0,C 180,E1 -6946.18,E2 -6946.18} C_VEL
LIN {X 0,Y 482.269,Z 420.197,A -85,B 0,C 180,E1 -6946.536,E2 -6946.536} C_VEL
LIN {X 0,Y 482.922,Z 402.189,A -85,B 0,C 180,E1 -6949.555,E2 -6949.555} C_VEL
LIN {X 0,Y 483.703,Z 383.916,A -85,B 0,C 180,E1 -6952.645,E2 -6952.645} C_VEL
LIN {X 0,Y 483.797,Z 377.404,A -85,B 0,C 180,E1 -6953.767,E2 -6953.767} C_VEL
LIN {X 0,Y 481.75,Z 366.48,A -85,B 0,C 180,E1 -6955.82,E2 -6955.82} C_VEL
LIN {X 0,Y 481.678,Z 366.484,A -85,B 0,C 180,E1 -6958.903,E2 -6958.903} C_VEL
LIN {X 0,Y 481.658,Z 366.488,A -85,B 0,C 180,E1 -6962.189,E2 -6962.189} C_VEL
LIN {X 0,Y 481.692,Z 366.478,A -85,B 0,C 180,E1 -6964.681,E2 -6964.681} C_VEL
LIN {X 0,Y 481.654,Z 366.487,A -85,B 0,C 180,E1 -6968.007,E2 -6968.007} C_VEL
LIN {X 0,Y 481.66,Z 366.484,A -85,B 0,C 180,E1 -6971.04,E2 -6971.04} C_VEL
LIN {X 0,Y 481.655,Z 366.483,A -85,B 0,C 180,E1 -6974.359,E2 -6974.359} C_VEL
LIN {X 0,Y 481.684,Z 366.48,A -85,B 0,C 180,E1 -6976.845,E2 -6976.845} C_VEL
LIN {X 0,Y 481.684,Z 366.481,A -85,B 0,C 180,E1 -6980.06,E2 -6980.06} C_VEL
LIN {X 0,Y 481.624,Z 366.493,A -85,B 0,C 180,E1 -6983.253,E2 -6983.253} C_VEL
LIN {X 0,Y 481.703,Z 366.477,A -85,B 0,C 180,E1 -6986.329,E2 -6986.329} C_VEL
LIN {X 0,Y 481.652,Z 366.491,A -85,B 0,C 180,E1 -6989.415,E2 -6989.415} C_VEL
LIN {X 0,Y 481.695,Z 366.478,A -85,B 0,C 180,E1 -6992.168,E2 -6992.168} C_VEL
LIN {X 0,Y 481.712,Z 366.48,A -85,B 0,C 180,E1 -6994.97,E2 -6994.97} C_VEL
LIN {X 0,Y 481.652,Z 366.486,A -85,B 0,C 180,E1 -6997.705,E2 -6997.705} C_VEL
LIN {X 0,Y 481.7,Z 366.478,A -85,B 0,C 180,E1 -7000.393,E2 -7000.393} C_VEL
LIN {X 0,Y 481.684,Z 366.486,A -85,B 0,C 180,E1 -7003.034,E2 -7003.034} C_VEL
LIN {X 0,Y 481.682,Z 366.482,A -85,B 0,C 180,E1 -7005.638,E2 -7005.638} C_VEL
LIN {X 0,Y 481.788,Z 366.467,A -85,B 0,C 180,E1 -7008.216,E2 -7008.216} C_VEL
LIN {X 0,Y 481.755,Z 366.472,A -85,B 0,C 180,E1 -7011.612,E2 -7011.612} C_VEL
LIN {X 0,Y 481.808,Z 366.464,A -85,B 0,C 180,E1 -7014.14,E2 -7014.14} C_VEL
LIN {X 0,Y 481.921,Z 366.452,A -85,B 0,C 180,E1 -7017.493,E2 -7017.493} C_VEL
LIN {X 0,Y 481.931,Z 366.449,A -85,B 0,C 180,E1 -7020,E2 -7020} C_VEL
LIN {X 0,Y 481.921,Z 366.453,A -85,B 0,C 180,E1 -7022.508,E2 -7022.508} C_VEL
LIN {X 0,Y 481.813,Z 366.463,A -85,B 0,C 180,E1 -7025.861,E2 -7025.861} C_VEL
LIN {X 0,Y 481.755,Z 366.473,A -85,B 0,C 180,E1 -7028.389,E2 -7028.389} C_VEL
LIN {X 0,Y 481.786,Z 366.467,A -85,B 0,C 180,E1 -7031.784,E2 -7031.784} C_VEL
LIN {X 0,Y 481.735,Z 366.475,A -85,B 0,C 180,E1 -7035.225,E2 -7035.225} C_VEL
LIN {X 0,Y 481.704,Z 366.485,A -85,B 0,C 180,E1 -7038.722,E2 -7038.722} C_VEL
LIN {X 0,Y 481.646,Z 366.485,A -85,B 0,C 180,E1 -7041.395,E2 -7041.395} C_VEL
LIN {X 0,Y 481.675,Z 366.483,A -85,B 0,C 180,E1 -7044.113,E2 -7044.113} C_VEL
LIN {X 0,Y 481.745,Z 366.474,A -85,B 0,C 180,E1 -7047.141,E2 -7047.141} C_VEL
LIN {X 0,Y 481.672,Z 366.481,A -85,B 0,C 180,E1 -7049.742,E2 -7049.742} C_VEL
LIN {X 0,Y 481.667,Z 366.488,A -85,B 0,C 180,E1 -7052.675,E2 -7052.675} C_VEL
LIN {X 0,Y 481.636,Z 366.486,A -85,B 0,C 180,E1 -7055.71,E2 -7055.71} C_VEL
LIN {X 0,Y 481.709,Z 366.476,A -85,B 0,C 180,E1 -7059.355,E2 -7059.355} C_VEL
LIN {X 0,Y 481.669,Z 366.487,A -85,B 0,C 180,E1 -7062.159,E2 -7062.159} C_VEL
LIN {X 0,Y 481.656,Z 366.49,A -85,B 0,C 180,E1 -7064.458,E2 -7064.458} C_VEL
LIN {X 0,Y 481.644,Z 366.487,A -85,B 0,C 180,E1 -7067.84,E2 -7067.84} C_VEL
LIN {X 0,Y 481.678,Z 366.483,A -85,B 0,C 180,E1 -7070.652,E2 -7070.652} C_VEL
LIN {X 0,Y 481.63,Z 366.486,A -85,B 0,C 180,E1 -7073.376,E2 -7073.376} C_VEL
LIN {X 0,Y 481.709,Z 366.483,A -85,B 0,C 180,E1 -7076.331,E2 -7076.331} C_VEL
LIN {X 0,Y 481.651,Z 366.484,A -85,B 0,C 180,E1 -7079.418,E2 -7079.418} C_VEL
LIN {X 0,Y 481.701,Z 366.485,A -85,B 0,C 180,E1 -7082.169,E2 -7082.169} C_VEL
LIN {X 0,Y 481.694,Z 366.482,A -85,B 0,C 180,E1 -7084.969,E2 -7084.969} C_VEL
LIN {X 0,Y 481.636,Z 366.491,A -85,B 0,C 180,E1 -7088.001,E2 -7088.001} C_VEL
LIN {X 0,Y 481.375,Z 366.81,A -85,B 0,C 180,E1 -7088.464,E2 -7088.464} C_VEL
LIN {X 0,Y 480.298,Z 368.256,A -85,B 0,C 180,E1 -7089.135,E2 -7089.135} C_VEL
LIN {X 0,Y 478.808,Z 370.507,A -85,B 0,C 180,E1 -7089.769,E2 -7089.769} C_VEL
LIN {X 0,Y 476.121,Z 376.361,A -85,B 0,C 180,E1 -7091.015,E2 -7091.015} C_VEL
LIN {X 0,Y 475.788,Z 378.361,A -85,B 0,C 180,E1 -7091.438,E2 -7091.438} C_VEL
LIN {X 0,Y 475.417,Z 387.001,A -85,B 0,C 180,E1 -7093.296,E2 -7093.296} C_VEL
LIN {X 0,Y 478.177,Z 400.592,A -85,B 0,C 180,E1 -7093.616,E2 -7093.616} C_VEL
LIN {X 0,Y 477.532,Z 494.037,A -85,B 0,C 180,E1 -7095.048,E2 -7095.048} C_VEL
LIN {X 0,Y 477.194,Z 507.911,A -85,B 0,C 180,E1 -7095.446,E2 -7095.446} C_VEL
LIN {X 0,Y 476.911,Z 520.315,A -85,B 0,C 180,E1 -7095.982,E2 -7095.982} C_VEL
LIN {X 0,Y 476.519,Z 531.754,A -85,B 0,C 180,E1 -7096.649,E2 -7096.649} C_VEL
LIN {X 0,Y 476.065,Z 543.521,A -85,B 0,C 180,E1 -7097.532,E2 -7097.532} C_VEL
LIN {X 0,Y 475.544,Z 553.755,A -85,B 0,C 180,E1 -7098.492,E2 -7098.492} C_VEL
LIN {X 0,Y 475.125,Z 562.932,A -85,B 0,C 180,E1 -7099.561,E2 -7099.561} C_VEL
LIN {X 0,Y 474.683,Z 571.839,A -85,B 0,C 180,E1 -7100.842,E2 -7100.842} C_VEL
LIN {X 0,Y 474.344,Z 579.008,A -85,B 0,C 180,E1 -7102.123,E2 -7102.123} C_VEL
LIN {X 0,Y 474.11,Z 585.416,A -85,B 0,C 180,E1 -7103.585,E2 -7103.585} C_VEL
LIN {X 0,Y 473.86,Z 589.856,A -85,B 0,C 180,E1 -7104.895,E2 -7104.895} C_VEL
LIN {X 0,Y 473.915,Z 592.135,A -85,B 0,C 180,E1 -7105.748,E2 -7105.748} C_VEL
LIN {X 0,Y 473.845,Z 593.995,A -85,B 0,C 180,E1 -7106.599,E2 -7106.599} C_VEL
LIN {X 0,Y 473.785,Z 595.397,A -85,B 0,C 180,E1 -7107.449,E2 -7107.449} C_VEL
LIN {X 0,Y 473.758,Z 596.393,A -85,B 0,C 180,E1 -7108.3,E2 -7108.3} C_VEL
LIN {X 0,Y 473.672,Z 597.245,A -85,B 0,C 180,E1 -7110,E2 -7110} C_VEL
LIN {X 0,Y 473.689,Z 597.059,A -85,B 0,C 180,E1 -7110.85,E2 -7110.85} C_VEL
LIN {X 0,Y 473.759,Z 596.475,A -85,B 0,C 180,E1 -7111.7,E2 -7111.7} C_VEL
LIN {X 0,Y 473.846,Z 594.16,A -85,B 0,C 180,E1 -7113.401,E2 -7113.401} C_VEL
LIN {X 0,Y 473.877,Z 591.305,A -85,B 0,C 180,E1 -7114.679,E2 -7114.679} C_VEL
LIN {X 0,Y 474.086,Z 587.426,A -85,B 0,C 180,E1 -7115.956,E2 -7115.956} C_VEL
LIN {X 0,Y 474.218,Z 582.428,A -85,B 0,C 180,E1 -7117.237,E2 -7117.237} C_VEL
LIN {X 0,Y 474.459,Z 576.134,A -85,B 0,C 180,E1 -7118.518,E2 -7118.518} C_VEL
LIN {X 0,Y 474.849,Z 568.249,A -85,B 0,C 180,E1 -7119.8,E2 -7119.8} C_VEL
LIN {X 0,Y 475.245,Z 558.441,A -85,B 0,C 180,E1 -7121.084,E2 -7121.084} C_VEL
LIN {X 0,Y 475.853,Z 548.143,A -85,B 0,C 180,E1 -7122.149,E2 -7122.149} C_VEL
LIN {X 0,Y 476.257,Z 536.617,A -85,B 0,C 180,E1 -7123.107,E2 -7123.107} C_VEL
LIN {X 0,Y 476.739,Z 524.966,A -85,B 0,C 180,E1 -7123.86,E2 -7123.86} C_VEL
LIN {X 0,Y 477.138,Z 512.937,A -85,B 0,C 180,E1 -7124.446,E2 -7124.446} C_VEL
LIN {X 0,Y 477.451,Z 499.836,A -85,B 0,C 180,E1 -7124.9,E2 -7124.9} C_VEL
LIN {X 0,Y 477.559,Z 487.234,A -85,B 0,C 180,E1 -7125.169,E2 -7125.169} C_VEL
LIN {X 0,Y 478.197,Z 400.749,A -85,B 0,C 180,E1 -7126.472,E2 -7126.472} C_VEL
LIN {X 0,Y 475.436,Z 387.001,A -85,B 0,C 180,E1 -7126.797,E2 -7126.797} C_VEL
LIN {X 0,Y 475.919,Z 374.913,A -85,B 0,C 180,E1 -7129.405,E2 -7129.405} C_VEL
LIN {X 0,Y 474.613,Z 367.369,A -85,B 0,C 180,E1 -7131.17,E2 -7131.17} C_VEL
LIN {X 0,Y 474.661,Z 367.362,A -85,B 0,C 180,E1 -7134.492,E2 -7134.492} C_VEL
LIN {X 0,Y 474.681,Z 367.353,A -85,B 0,C 180,E1 -7137.334,E2 -7137.334} C_VEL
LIN {X 0,Y 474.605,Z 367.366,A -85,B 0,C 180,E1 -7140.229,E2 -7140.229} C_VEL
LIN {X 0,Y 474.642,Z 367.358,A -85,B 0,C 180,E1 -7143.219,E2 -7143.219} C_VEL
LIN {X 0,Y 474.592,Z 367.366,A -85,B 0,C 180,E1 -7146.322,E2 -7146.322} C_VEL
LIN {X 0,Y 474.625,Z 367.365,A -85,B 0,C 180,E1 -7149.647,E2 -7149.647} C_VEL
LIN {X 0,Y 474.611,Z 367.361,A -85,B 0,C 180,E1 -7152.933,E2 -7152.933} C_VEL
LIN {X 0,Y 474.614,Z 367.366,A -85,B 0,C 180,E1 -7155.895,E2 -7155.895} C_VEL
LIN {X 0,Y 474.641,Z 367.358,A -85,B 0,C 180,E1 -7159.037,E2 -7159.037} C_VEL
LIN {X 0,Y 474.611,Z 367.368,A -85,B 0,C 180,E1 -7161.702,E2 -7161.702} C_VEL
LIN {X 0,Y 474.625,Z 367.359,A -85,B 0,C 180,E1 -7164.725,E2 -7164.725} C_VEL
LIN {X 0,Y 474.631,Z 367.363,A -85,B 0,C 180,E1 -7167.787,E2 -7167.787} C_VEL
LIN {X 0,Y 474.617,Z 367.361,A -85,B 0,C 180,E1 -7170.884,E2 -7170.884} C_VEL
LIN {X 0,Y 474.66,Z 367.361,A -85,B 0,C 180,E1 -7173.628,E2 -7173.628} C_VEL
LIN {X 0,Y 474.629,Z 367.359,A -85,B 0,C 180,E1 -7176.64,E2 -7176.64} C_VEL
LIN {X 0,Y 474.649,Z 367.357,A -85,B 0,C 180,E1 -7180.089,E2 -7180.089} C_VEL
LIN {X 0,Y 474.643,Z 367.358,A -85,B 0,C 180,E1 -7182.774,E2 -7182.774} C_VEL
LIN {X 0,Y 474.643,Z 367.363,A -85,B 0,C 180,E1 -7185.421,E2 -7185.421} C_VEL
LIN {X 0,Y 474.73,Z 367.346,A -85,B 0,C 180,E1 -7188.038,E2 -7188.038} C_VEL
LIN {X 0,Y 474.72,Z 367.352,A -85,B 0,C 180,E1 -7191.486,E2 -7191.486} C_VEL
LIN {X 0,Y 474.771,Z 367.341,A -85,B 0,C 180,E1 -7194.052,E2 -7194.052} C_VEL
LIN {X 0,Y 474.887,Z 367.33,A -85,B 0,C 180,E1 -7197.455,E2 -7197.455} C_VEL
LIN {X 0,Y 474.869,Z 367.333,A -85,B 0,C 180,E1 -7200.848,E2 -7200.848} C_VEL
LIN {X 0,Y 474.887,Z 367.328,A -85,B 0,C 180,E1 -7202.545,E2 -7202.545} C_VEL
LIN {X 0,Y 474.775,Z 367.34,A -85,B 0,C 180,E1 -7205.948,E2 -7205.948} C_VEL
LIN {X 0,Y 474.721,Z 367.349,A -85,B 0,C 180,E1 -7208.514,E2 -7208.514} C_VEL
LIN {X 0,Y 474.73,Z 367.346,A -85,B 0,C 180,E1 -7211.962,E2 -7211.962} C_VEL
LIN {X 0,Y 474.672,Z 367.353,A -85,B 0,C 180,E1 -7215.768,E2 -7215.768} C_VEL
LIN {X 0,Y 474.657,Z 367.361,A -85,B 0,C 180,E1 -7219.011,E2 -7219.011} C_VEL
LIN {X 0,Y 474.59,Z 367.363,A -85,B 0,C 180,E1 -7221.729,E2 -7221.729} C_VEL
LIN {X 0,Y 474.654,Z 367.36,A -85,B 0,C 180,E1 -7224.493,E2 -7224.493} C_VEL
LIN {X 0,Y 474.692,Z 367.352,A -85,B 0,C 180,E1 -7227.339,E2 -7227.339} C_VEL
LIN {X 0,Y 474.598,Z 367.369,A -85,B 0,C 180,E1 -7230.811,E2 -7230.811} C_VEL
LIN {X 0,Y 474.632,Z 367.359,A -85,B 0,C 180,E1 -7233.985,E2 -7233.985} C_VEL
LIN {X 0,Y 474.57,Z 367.37,A -85,B 0,C 180,E1 -7236.901,E2 -7236.901} C_VEL
LIN {X 0,Y 474.645,Z 367.356,A -85,B 0,C 180,E1 -7239.652,E2 -7239.652} C_VEL
LIN {X 0,Y 474.648,Z 367.359,A -85,B 0,C 180,E1 -7242.931,E2 -7242.931} C_VEL
LIN {X 0,Y 474.611,Z 367.362,A -85,B 0,C 180,E1 -7245.897,E2 -7245.897} C_VEL
LIN {X 0,Y 474.629,Z 367.359,A -85,B 0,C 180,E1 -7249.041,E2 -7249.041} C_VEL
LIN {X 0,Y 474.608,Z 367.362,A -85,B 0,C 180,E1 -7251.705,E2 -7251.705} C_VEL
LIN {X 0,Y 474.629,Z 367.361,A -85,B 0,C 180,E1 -7254.727,E2 -7254.727} C_VEL
LIN {X 0,Y 474.637,Z 367.36,A -85,B 0,C 180,E1 -7257.789,E2 -7257.789} C_VEL
LIN {X 0,Y 474.624,Z 367.363,A -85,B 0,C 180,E1 -7260.885,E2 -7260.885} C_VEL
LIN {X 0,Y 474.701,Z 367.358,A -85,B 0,C 180,E1 -7263.982,E2 -7263.982} C_VEL
LIN {X 0,Y 476.882,Z 379.021,A -85,B 0,C 180,E1 -7266.191,E2 -7266.191} C_VEL
LIN {X 0,Y 476.381,Z 392.831,A -85,B 0,C 180,E1 -7268.585,E2 -7268.585} C_VEL
LIN {X 0,Y 475.594,Z 412.352,A -85,B 0,C 180,E1 -7271.922,E2 -7271.922} C_VEL
LIN {X 0,Y 475.32,Z 420.016,A -85,B 0,C 180,E1 -7273.23,E2 -7273.23} C_VEL
LIN {X 0,Y 478.048,Z 438.3,A -85,B 0,C 180,E1 -7273.614,E2 -7273.614} C_VEL
LIN {X 0,Y 477.39,Z 528.386,A -85,B 0,C 180,E1 -7274.989,E2 -7274.989} C_VEL
LIN {X 0,Y 477.04,Z 541.663,A -85,B 0,C 180,E1 -7275.36,E2 -7275.36} C_VEL
LIN {X 0,Y 476.57,Z 554.957,A -85,B 0,C 180,E1 -7275.917,E2 -7275.917} C_VEL
LIN {X 0,Y 476.181,Z 566.123,A -85,B 0,C 180,E1 -7276.559,E2 -7276.559} C_VEL
LIN {X 0,Y 475.631,Z 577.312,A -85,B 0,C 180,E1 -7277.377,E2 -7277.377} C_VEL
LIN {X 0,Y 475.211,Z 588.189,A -85,B 0,C 180,E1 -7278.375,E2 -7278.375} C_VEL
LIN {X 0,Y 474.794,Z 596.741,A -85,B 0,C 180,E1 -7279.338,E2 -7279.338} C_VEL
LIN {X 0,Y 474.457,Z 604.634,A -85,B 0,C 180,E1 -7280.408,E2 -7280.408} C_VEL
LIN {X 0,Y 474.166,Z 612.346,A -85,B 0,C 180,E1 -7281.691,E2 -7281.691} C_VEL
LIN {X 0,Y 473.935,Z 619.458,A -85,B 0,C 180,E1 -7283.187,E2 -7283.187} C_VEL
LIN {X 0,Y 473.846,Z 624.191,A -85,B 0,C 180,E1 -7284.468,E2 -7284.468} C_VEL
LIN {X 0,Y 473.735,Z 627.806,A -85,B 0,C 180,E1 -7285.746,E2 -7285.746} C_VEL
LIN {X 0,Y 473.795,Z 629.675,A -85,B 0,C 180,E1 -7286.599,E2 -7286.599} C_VEL
LIN {X 0,Y 473.724,Z 632.071,A -85,B 0,C 180,E1 -7288.3,E2 -7288.3} C_VEL
LIN {X 0,Y 473.688,Z 632.679,A -85,B 0,C 180,E1 -7289.15,E2 -7289.15} C_VEL
LIN {X 0,Y 473.67,Z 632.895,A -85,B 0,C 180,E1 -7290,E2 -7290} C_VEL
LIN {X 0,Y 473.688,Z 632.68,A -85,B 0,C 180,E1 -7290.85,E2 -7290.85} C_VEL
LIN {X 0,Y 473.724,Z 632.072,A -85,B 0,C 180,E1 -7291.7,E2 -7291.7} C_VEL
LIN {X 0,Y 473.795,Z 629.678,A -85,B 0,C 180,E1 -7293.401,E2 -7293.401} C_VEL
LIN {X 0,Y 473.763,Z 626.734,A -85,B 0,C 180,E1 -7294.68,E2 -7294.68} C_VEL
LIN {X 0,Y 473.836,Z 622.752,A -85,B 0,C 180,E1 -7295.959,E2 -7295.959} C_VEL
LIN {X 0,Y 474.016,Z 616.631,A -85,B 0,C 180,E1 -7297.454,E2 -7297.454} C_VEL
LIN {X 0,Y 474.27,Z 609.943,A -85,B 0,C 180,E1 -7298.736,E2 -7298.736} C_VEL
LIN {X 0,Y 474.569,Z 601.645,A -85,B 0,C 180,E1 -7300.021,E2 -7300.021} C_VEL
LIN {X 0,Y 474.996,Z 593.146,A -85,B 0,C 180,E1 -7301.09,E2 -7301.09} C_VEL
LIN {X 0,Y 475.472,Z 582.907,A -85,B 0,C 180,E1 -7302.135,E2 -7302.135} C_VEL
LIN {X 0,Y 475.864,Z 572.546,A -85,B 0,C 180,E1 -7302.994,E2 -7302.994} C_VEL
LIN {X 0,Y 476.363,Z 560.875,A -85,B 0,C 180,E1 -7303.762,E2 -7303.762} C_VEL
LIN {X 0,Y 476.793,Z 549.204,A -85,B 0,C 180,E1 -7304.348,E2 -7304.348} C_VEL
LIN {X 0,Y 477.193,Z 536.675,A -85,B 0,C 180,E1 -7304.799,E2 -7304.799} C_VEL
LIN {X 0,Y 477.488,Z 524.001,A -85,B 0,C 180,E1 -7305.09,E2 -7305.09} C_VEL
LIN {X 0,Y 477.933,Z 437.246,A -85,B 0,C 180,E1 -7306.405,E2 -7306.405} C_VEL
LIN {X 0,Y 475.307,Z 419.993,A -85,B 0,C 180,E1 -7306.775,E2 -7306.775} C_VEL
LIN {X 0,Y 475.922,Z 403.374,A -85,B 0,C 180,E1 -7309.607,E2 -7309.607} C_VEL
LIN {X 0,Y 476.76,Z 384.987,A -85,B 0,C 180,E1 -7312.765,E2 -7312.765} C_VEL
LIN {X 0,Y 476.787,Z 378.241,A -85,B 0,C 180,E1 -7313.949,E2 -7313.949} C_VEL
LIN {X 0,Y 474.701,Z 367.358,A -85,B 0,C 180,E1 -7316.018,E2 -7316.018} C_VEL
LIN {X 0,Y 474.646,Z 367.362,A -85,B 0,C 180,E1 -7318.282,E2 -7318.282} C_VEL
LIN {X 0,Y 474.6,Z 367.368,A -85,B 0,C 180,E1 -7321.217,E2 -7321.217} C_VEL
LIN {X 0,Y 474.632,Z 367.36,A -85,B 0,C 180,E1 -7324.24,E2 -7324.24} C_VEL
LIN {X 0,Y 474.59,Z 367.368,A -85,B 0,C 180,E1 -7327.383,E2 -7327.383} C_VEL
LIN {X 0,Y 474.625,Z 367.367,A -85,B 0,C 180,E1 -7329.647,E2 -7329.647} C_VEL
LIN {X 0,Y 474.632,Z 367.359,A -85,B 0,C 180,E1 -7332.931,E2 -7332.931} C_VEL
LIN {X 0,Y 474.614,Z 367.364,A -85,B 0,C 180,E1 -7335.895,E2 -7335.895} C_VEL
LIN {X 0,Y 474.641,Z 367.359,A -85,B 0,C 180,E1 -7339.037,E2 -7339.037} C_VEL
LIN {X 0,Y 474.611,Z 367.366,A -85,B 0,C 180,E1 -7341.702,E2 -7341.702} C_VEL
LIN {X 0,Y 474.624,Z 367.36,A -85,B 0,C 180,E1 -7344.726,E2 -7344.726} C_VEL
LIN {X 0,Y 474.631,Z 367.361,A -85,B 0,C 180,E1 -7347.787,E2 -7347.787} C_VEL
LIN {X 0,Y 474.625,Z 367.361,A -85,B 0,C 180,E1 -7350.882,E2 -7350.882} C_VEL
LIN {X 0,Y 474.659,Z 367.358,A -85,B 0,C 180,E1 -7353.628,E2 -7353.628} C_VEL
LIN {X 0,Y 474.628,Z 367.36,A -85,B 0,C 180,E1 -7356.641,E2 -7356.641} C_VEL
LIN {X 0,Y 474.649,Z 367.356,A -85,B 0,C 180,E1 -7360.089,E2 -7360.089} C_VEL
LIN {X 0,Y 474.643,Z 367.36,A -85,B 0,C 180,E1 -7362.774,E2 -7362.774} C_VEL
LIN {X 0,Y 474.641,Z 367.361,A -85,B 0,C 180,E1 -7365.421,E2 -7365.421} C_VEL
LIN {X 0,Y 474.73,Z 367.346,A -85,B 0,C 180,E1 -7368.038,E2 -7368.038} C_VEL
LIN {X 0,Y 474.72,Z 367.35,A -85,B 0,C 180,E1 -7371.486,E2 -7371.486} C_VEL
LIN {X 0,Y 474.771,Z 367.341,A -85,B 0,C 180,E1 -7374.052,E2 -7374.052} C_VEL
LIN {X 0,Y 474.887,Z 367.329,A -85,B 0,C 180,E1 -7377.455,E2 -7377.455} C_VEL
LIN {X 0,Y 474.869,Z 367.336,A -85,B 0,C 180,E1 -7380.848,E2 -7380.848} C_VEL
LIN {X 0,Y 474.887,Z 367.33,A -85,B 0,C 180,E1 -7382.545,E2 -7382.545} C_VEL
LIN {X 0,Y 474.775,Z 367.34,A -85,B 0,C 180,E1 -7385.948,E2 -7385.948} C_VEL
LIN {X 0,Y 474.72,Z 367.351,A -85,B 0,C 180,E1 -7388.514,E2 -7388.514} C_VEL
LIN {X 0,Y 474.73,Z 367.346,A -85,B 0,C 180,E1 -7391.962,E2 -7391.962} C_VEL
LIN {X 0,Y 474.672,Z 367.353,A -85,B 0,C 180,E1 -7395.768,E2 -7395.768} C_VEL
LIN {X 0,Y 474.657,Z 367.359,A -85,B 0,C 180,E1 -7399.011,E2 -7399.011} C_VEL
LIN {X 0,Y 474.59,Z 367.363,A -85,B 0,C 180,E1 -7401.729,E2 -7401.729} C_VEL
LIN {X 0,Y 474.655,Z 367.362,A -85,B 0,C 180,E1 -7404.493,E2 -7404.493} C_VEL
LIN {X 0,Y 474.692,Z 367.351,A -85,B 0,C 180,E1 -7407.339,E2 -7407.339} C_VEL
LIN {X 0,Y 474.599,Z 367.367,A -85,B 0,C 180,E1 -7410.811,E2 -7410.811} C_VEL
LIN {X 0,Y 474.632,Z 367.36,A -85,B 0,C 180,E1 -7413.985,E2 -7413.985} C_VEL
LIN {X 0,Y 474.569,Z 367.368,A -85,B 0,C 180,E1 -7416.901,E2 -7416.901} C_VEL
LIN {X 0,Y 474.646,Z 367.357,A -85,B 0,C 180,E1 -7419.652,E2 -7419.652} C_VEL
LIN {X 0,Y 474.647,Z 367.358,A -85,B 0,C 180,E1 -7422.931,E2 -7422.931} C_VEL
LIN {X 0,Y 474.606,Z 367.364,A -85,B 0,C 180,E1 -7425.896,E2 -7425.896} C_VEL
LIN {X 0,Y 474.625,Z 367.359,A -85,B 0,C 180,E1 -7429.042,E2 -7429.042} C_VEL
LIN {X 0,Y 474.609,Z 367.363,A -85,B 0,C 180,E1 -7431.705,E2 -7431.705} C_VEL
LIN {X 0,Y 474.629,Z 367.36,A -85,B 0,C 180,E1 -7434.727,E2 -7434.727} C_VEL
LIN {X 0,Y 474.635,Z 367.361,A -85,B 0,C 180,E1 -7437.789,E2 -7437.789} C_VEL
LIN {X 0,Y 474.625,Z 367.359,A -85,B 0,C 180,E1 -7440.885,E2 -7440.885} C_VEL
LIN {X 0,Y 474.654,Z 367.358,A -85,B 0,C 180,E1 -7443.629,E2 -7443.629} C_VEL
LIN {X 0,Y 474.636,Z 367.363,A -85,B 0,C 180,E1 -7446.642,E2 -7446.642} C_VEL
LIN {X 0,Y 474.684,Z 367.557,A -85,B 0,C 180,E1 -7448.983,E2 -7448.983} C_VEL
LIN {X 0,Y 475.86,Z 374.498,A -85,B 0,C 180,E1 -7450.592,E2 -7450.592} C_VEL
